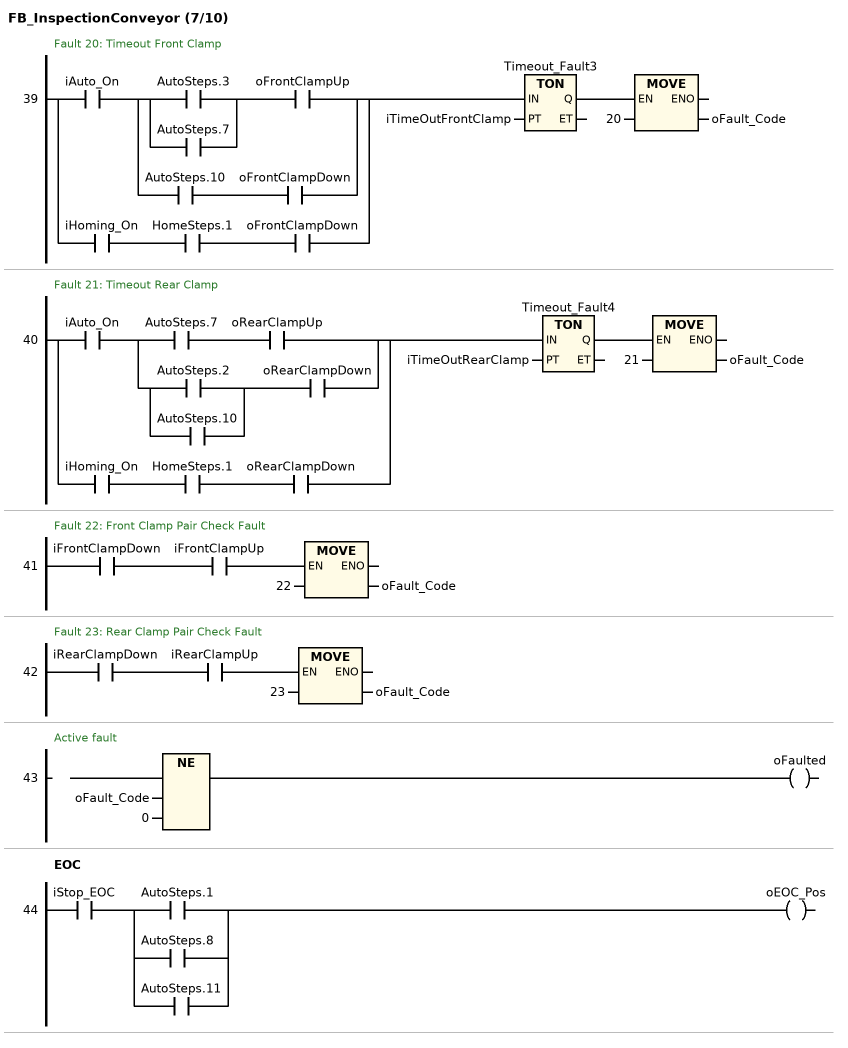
// NETWORK 39
// Fault 20: Timeout Front Clamp
Timeout_Fault3(IN := iAuto_On AND ((AutoSteps.3 OR AutoSteps.7) AND oFrontClampUp OR AutoSteps.10 AND oFrontClampDown) OR iHoming_On AND HomeSteps.1 AND oFrontClampDown, PT := iTimeOutFrontClamp); // TON
IF Timeout_Fault3.Q THEN oFault_Code := 20; END_IF

// NETWORK 40
// Fault 21: Timeout Rear Clamp
Timeout_Fault4(IN := iAuto_On AND (AutoSteps.7 AND oRearClampUp OR (AutoSteps.2 OR AutoSteps.10) AND oRearClampDown) OR iHoming_On AND HomeSteps.1 AND oRearClampDown, PT := iTimeOutRearClamp); // TON
IF Timeout_Fault4.Q THEN oFault_Code := 21; END_IF

// NETWORK 41
// Fault 22: Front Clamp Pair Check Fault
IF iFrontClampDown AND iFrontClampUp THEN oFault_Code := 22; END_IF

// NETWORK 42
// Fault 23: Rear Clamp Pair Check Fault
IF iRearClampDown AND iRearClampUp THEN oFault_Code := 23; END_IF

// NETWORK 43
// Active fault
oFaulted := oFault_Code <> 0;

// NETWORK 44: EOC
oEOC_Pos := iStop_EOC AND (AutoSteps.1 OR AutoSteps.8 OR AutoSteps.11);

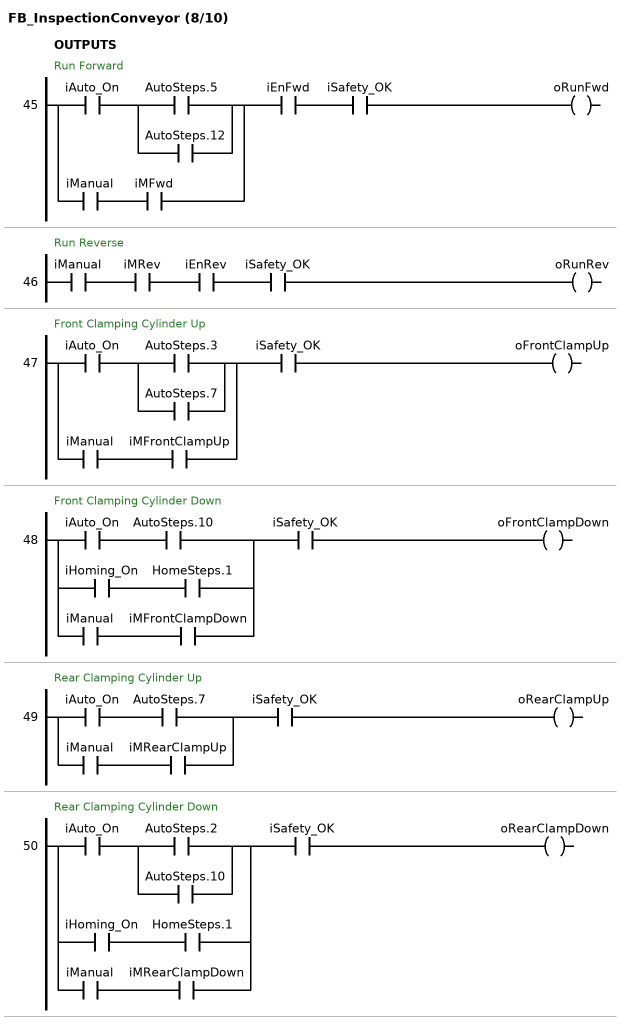
// NETWORK 45: OUTPUTS
// Run Forward
oRunFwd := (iAuto_On AND (AutoSteps.5 OR AutoSteps.12) OR iManual AND iMFwd) AND iEnFwd AND iSafety_OK;

// NETWORK 46
// Run Reverse
oRunRev := iManual AND iMRev AND iEnRev AND iSafety_OK;

// NETWORK 47
// Front Clamping Cylinder Up
oFrontClampUp := (iAuto_On AND (AutoSteps.3 OR AutoSteps.7) OR iManual AND iMFrontClampUp) AND iSafety_OK;

// NETWORK 48
// Front Clamping Cylinder Down
oFrontClampDown := (iAuto_On AND AutoSteps.10 OR iHoming_On AND HomeSteps.1 OR iManual AND iMFrontClampDown) AND iSafety_OK;

// NETWORK 49
// Rear Clamping Cylinder Up
oRearClampUp := (iAuto_On AND AutoSteps.7 OR iManual AND iMRearClampUp) AND iSafety_OK;

// NETWORK 50
// Rear Clamping Cylinder Down
oRearClampDown := (iAuto_On AND (AutoSteps.2 OR AutoSteps.10) OR iHoming_On AND HomeSteps.1 OR iManual AND iMRearClampDown) AND iSafety_OK;

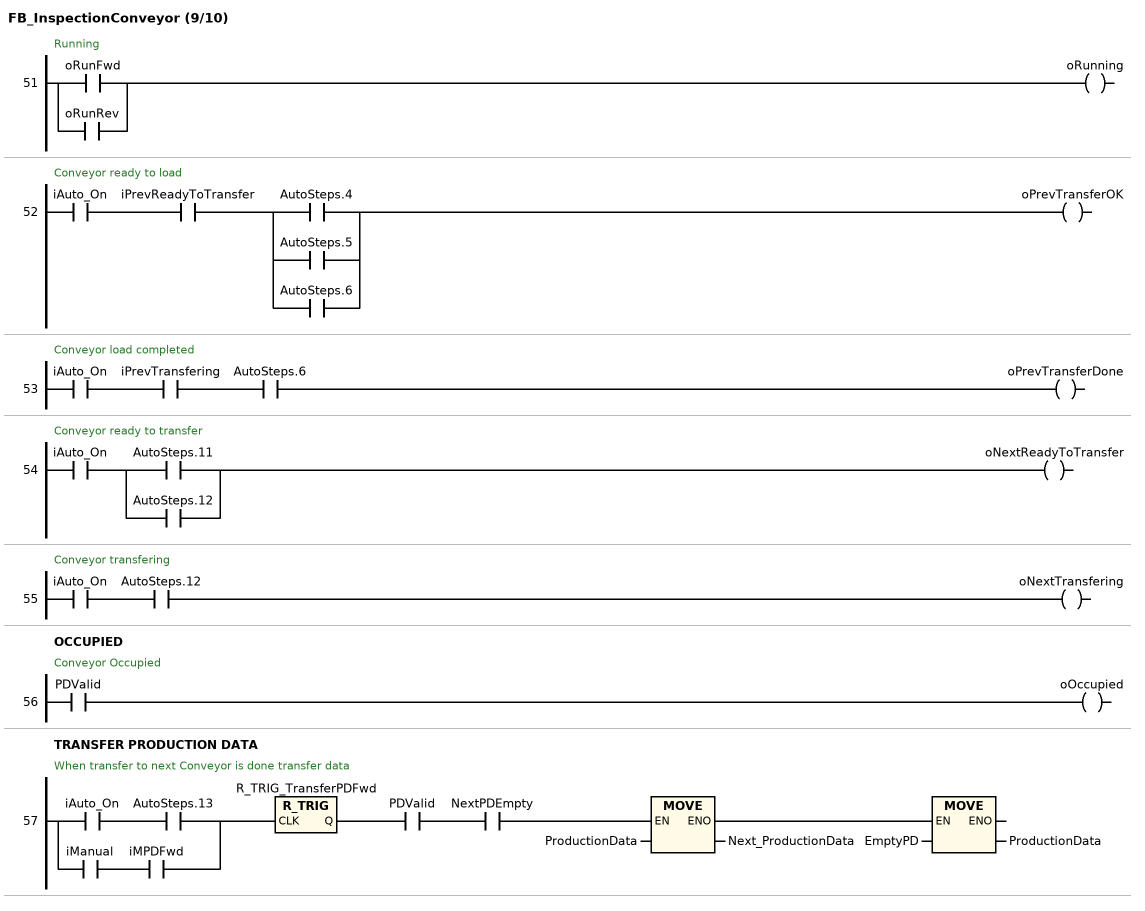
// NETWORK 51
// Running
oRunning := oRunFwd OR oRunRev;

// NETWORK 52
// Conveyor ready to load
oPrevTransferOK := iAuto_On AND iPrevReadyToTransfer AND (AutoSteps.4 OR AutoSteps.5 OR AutoSteps.6);

// NETWORK 53
// Conveyor load completed
oPrevTransferDone := iAuto_On AND iPrevTransfering AND AutoSteps.6;

// NETWORK 54
// Conveyor ready to transfer
oNextReadyToTransfer := iAuto_On AND (AutoSteps.11 OR AutoSteps.12);

// NETWORK 55
// Conveyor transfering
oNextTransfering := iAuto_On AND AutoSteps.12;

// NETWORK 56: OCCUPIED
// Conveyor Occupied
oOccupied := PDValid;

// NETWORK 57: TRANSFER PRODUCTION DATA
// When transfer to next Conveyor is done transfer data
R_TRIG_TransferPDFwd(CLK := iAuto_On AND AutoSteps.13 OR iManual AND iMPDFwd); // R_TRIG
_w20 := R_TRIG_TransferPDFwd.Q AND PDValid AND NextPDEmpty;
IF _w20 THEN Next_ProductionData := ProductionData; END_IF
IF _w20 THEN ProductionData := EmptyPD; END_IF

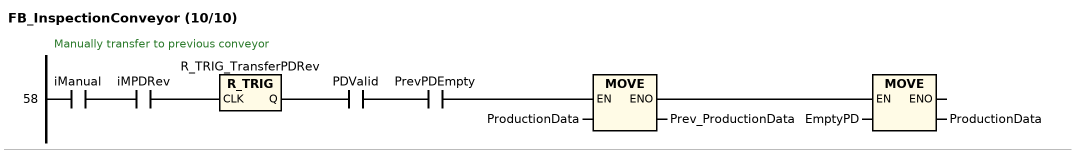
// NETWORK 58
// Manually transfer to previous conveyor
R_TRIG_TransferPDRev(CLK := iManual AND iMPDRev); // R_TRIG
_w21 := R_TRIG_TransferPDRev.Q AND PDValid AND PrevPDEmpty;
IF _w21 THEN Prev_ProductionData := ProductionData; END_IF
IF _w21 THEN ProductionData := EmptyPD; END_IF

END_FUNCTION_BLOCK

// Device/Application/FBs/Convert_RFID
FUNCTION Convert_RFID : STRING
VAR_INPUT
	iLecture: STRING := '';
	iID: UDINT := 0;
	iNumber: UINT := 0;
	iStatus: WORD := 0;
END_VAR
VAR_OUTPUT
	oID: UDINT;
	oNumber: UINT;
	oStatus: WORD;
END_VAR

oID := STRING_TO_UDINT(LEFT(iLecture, 4));
oNumber := STRING_TO_UINT(RIGHT(LEFT(iLecture, 8),4));
oStatus := STRING_TO_WORD(RIGHT(iLecture, 16));


Convert_RFID := CONCAT(UDINT_TO_STRING(iID),CONCAT(UINT_TO_STRING(iNumber),WORD_TO_STRING(iStatus)));

END_FUNCTION

// Device/Application/FBs/CombineData
PROGRAM CombineData
VAR_INPUT
	iCycleTime: STRING(1024);
	iProduct: STRING(1024);
END_VAR
VAR_OUTPUT
	oString: STRING(1024);
END_VAR

oString := CONCAT(iCycleTime,CONCAT('-',iProduct));

END_PROGRAM

// Device/Application/SOP630
PROGRAM SOP630
VAR
END_VAR

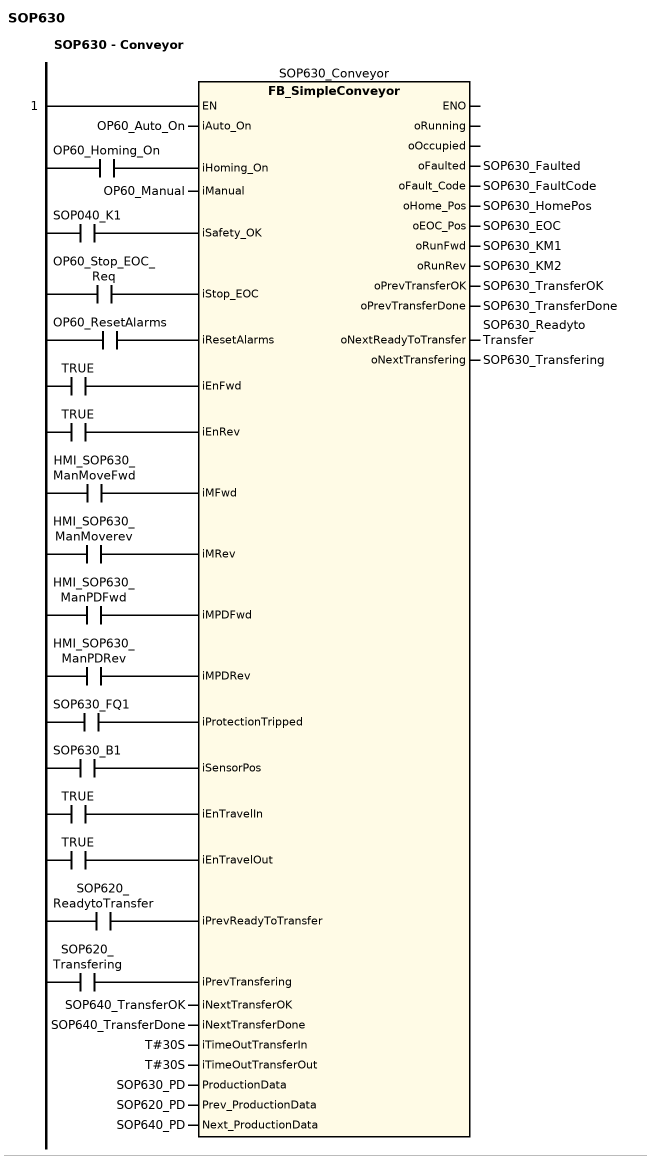
// NETWORK 1: SOP630 - Conveyor
SOP630_Conveyor(
    iAuto_On := OP60_Auto_On,
    iHoming_On := OP60_Homing_On,
    iManual := OP60_Manual,
    iSafety_OK := SOP040_K1,
    iStop_EOC := OP60_Stop_EOC_Req,
    iResetAlarms := OP60_ResetAlarms,
    iEnFwd := TRUE,
    iEnRev := TRUE,
    iMFwd := HMI_SOP630_ManMoveFwd,
    iMRev := HMI_SOP630_ManMoverev,
    iMPDFwd := HMI_SOP630_ManPDFwd,
    iMPDRev := HMI_SOP630_ManPDRev,
    iProtectionTripped := SOP630_FQ1,
    iSensorPos := SOP630_B1,
    iEnTravelIn := TRUE,
    iEnTravelOut := TRUE,
    iPrevReadyToTransfer := SOP620_ReadytoTransfer,
    iPrevTransfering := SOP620_Transfering,
    iNextTransferOK := SOP640_TransferOK,
    iNextTransferDone := SOP640_TransferDone,
    iTimeOutTransferIn := T#30S,
    iTimeOutTransferOut := T#30S,
    ProductionData := SOP630_PD,
    Prev_ProductionData := SOP620_PD,
    Next_ProductionData := SOP640_PD,
    oFaulted => SOP630_Faulted,
    oFault_Code => SOP630_FaultCode,
    oHome_Pos => SOP630_HomePos,
    oEOC_Pos => SOP630_EOC,
    oRunFwd => SOP630_KM1,
    oRunRev => SOP630_KM2,
    oPrevTransferOK => SOP630_TransferOK,
    oPrevTransferDone => SOP630_TransferDone,
    oNextReadyToTransfer => SOP630_ReadytoTransfer,
    oNextTransfering => SOP630_Transfering); // FB_SimpleConveyor

END_PROGRAM

// Device/Application/SOP620
PROGRAM SOP620
VAR
END_VAR

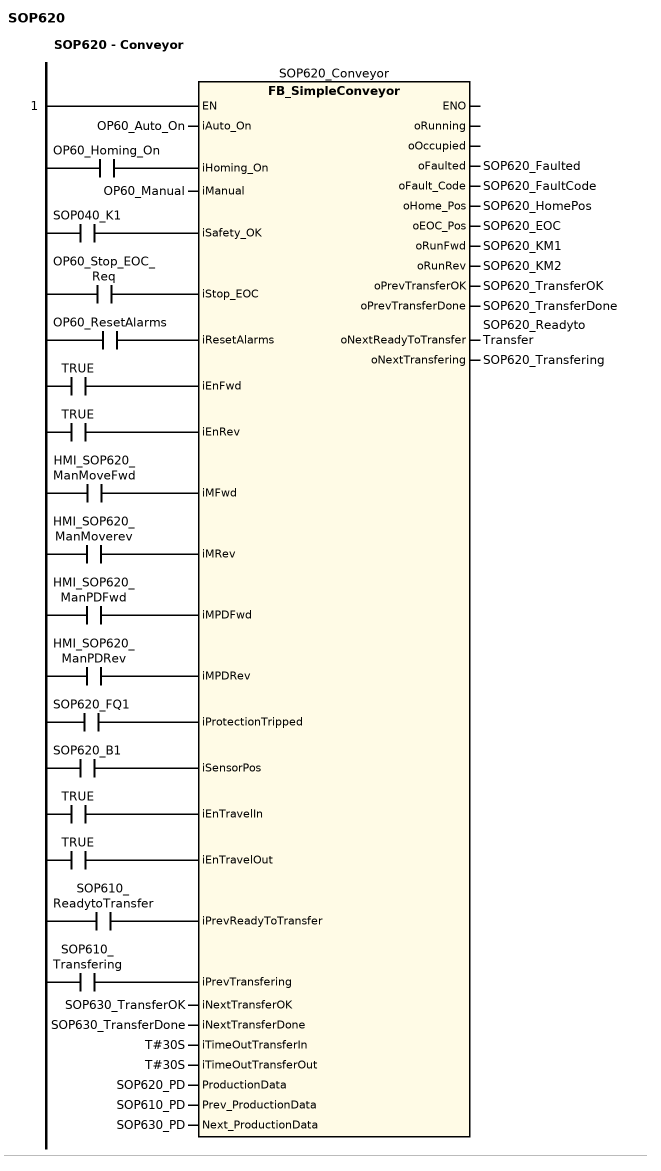
// NETWORK 1: SOP620 - Conveyor
SOP620_Conveyor(
    iAuto_On := OP60_Auto_On,
    iHoming_On := OP60_Homing_On,
    iManual := OP60_Manual,
    iSafety_OK := SOP040_K1,
    iStop_EOC := OP60_Stop_EOC_Req,
    iResetAlarms := OP60_ResetAlarms,
    iEnFwd := TRUE,
    iEnRev := TRUE,
    iMFwd := HMI_SOP620_ManMoveFwd,
    iMRev := HMI_SOP620_ManMoverev,
    iMPDFwd := HMI_SOP620_ManPDFwd,
    iMPDRev := HMI_SOP620_ManPDRev,
    iProtectionTripped := SOP620_FQ1,
    iSensorPos := SOP620_B1,
    iEnTravelIn := TRUE,
    iEnTravelOut := TRUE,
    iPrevReadyToTransfer := SOP610_ReadytoTransfer,
    iPrevTransfering := SOP610_Transfering,
    iNextTransferOK := SOP630_TransferOK,
    iNextTransferDone := SOP630_TransferDone,
    iTimeOutTransferIn := T#30S,
    iTimeOutTransferOut := T#30S,
    ProductionData := SOP620_PD,
    Prev_ProductionData := SOP610_PD,
    Next_ProductionData := SOP630_PD,
    oFaulted => SOP620_Faulted,
    oFault_Code => SOP620_FaultCode,
    oHome_Pos => SOP620_HomePos,
    oEOC_Pos => SOP620_EOC,
    oRunFwd => SOP620_KM1,
    oRunRev => SOP620_KM2,
    oPrevTransferOK => SOP620_TransferOK,
    oPrevTransferDone => SOP620_TransferDone,
    oNextReadyToTransfer => SOP620_ReadytoTransfer,
    oNextTransfering => SOP620_Transfering); // FB_SimpleConveyor

END_PROGRAM

// Device/Application/SOP610
PROGRAM SOP610
VAR
	ID_counter: UDINT := 1000;
	Check_not_empty_msg: BOOL;
END_VAR
VAR // added by the converter: edge detectors and wires of the graphical bodies
    _w1, _w2, _w3, _w4, _w5, _w6, _w7 : BOOL;
    _rt1, _rt2 : R_TRIG;
END_VAR

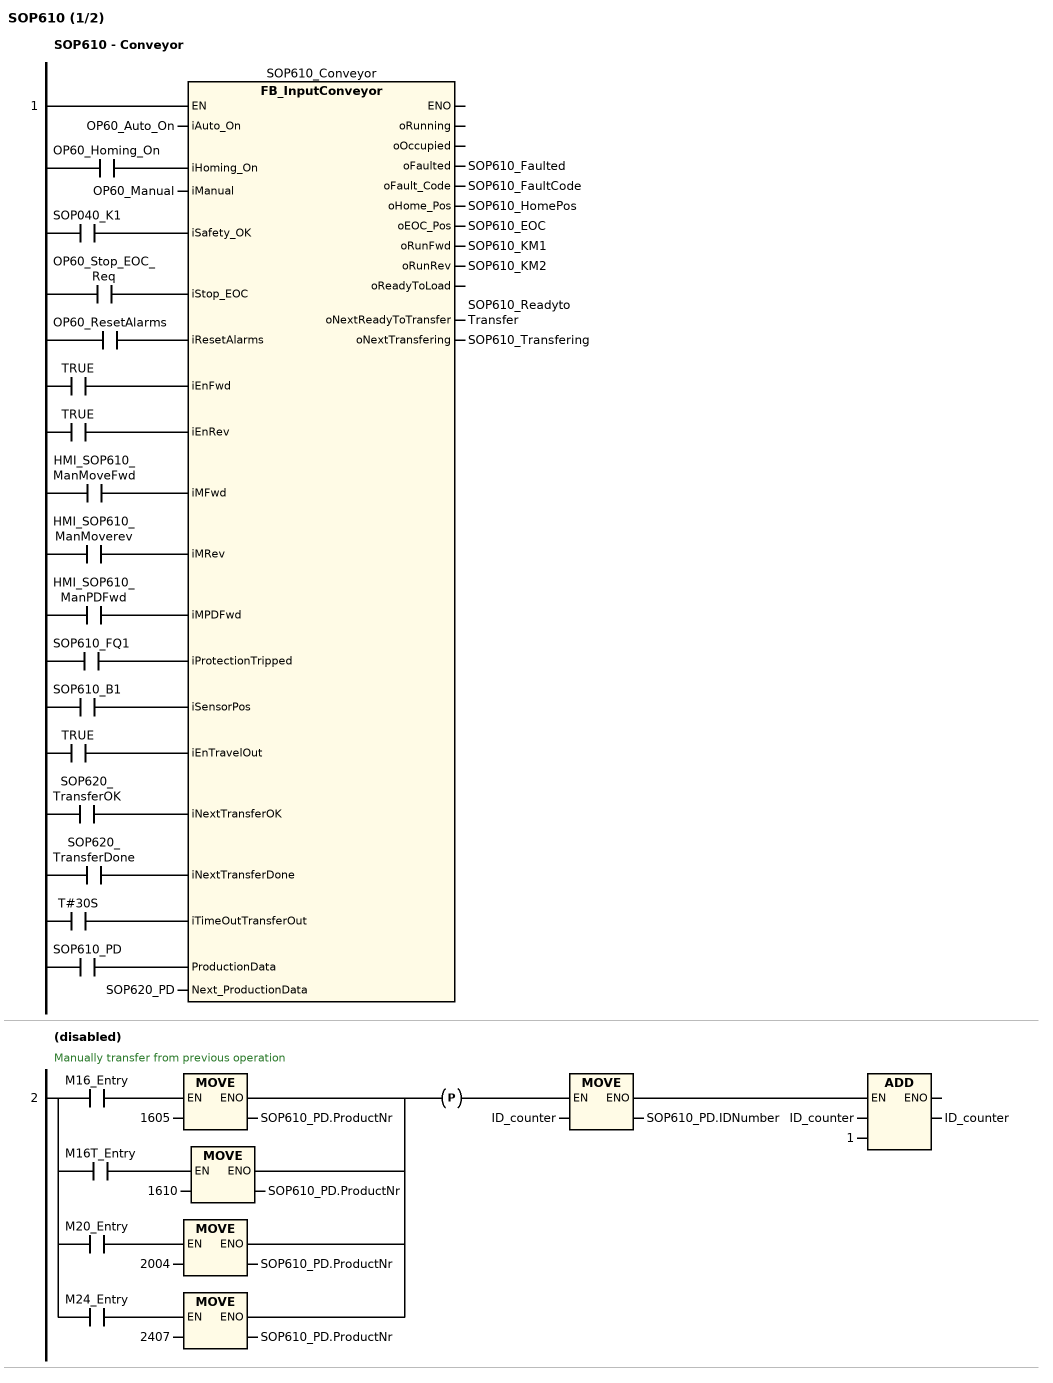
// NETWORK 1: SOP610 - Conveyor
SOP610_Conveyor(
    iAuto_On := OP60_Auto_On,
    iHoming_On := OP60_Homing_On,
    iManual := OP60_Manual,
    iSafety_OK := SOP040_K1,
    iStop_EOC := OP60_Stop_EOC_Req,
    iResetAlarms := OP60_ResetAlarms,
    iEnFwd := TRUE,
    iEnRev := TRUE,
    iMFwd := HMI_SOP610_ManMoveFwd,
    iMRev := HMI_SOP610_ManMoverev,
    iMPDFwd := HMI_SOP610_ManPDFwd,
    iProtectionTripped := SOP610_FQ1,
    iSensorPos := SOP610_B1,
    iEnTravelOut := TRUE,
    iNextTransferOK := SOP620_TransferOK,
    iNextTransferDone := SOP620_TransferDone,
    iTimeOutTransferOut := T#30S,
    ProductionData := SOP610_PD,
    Next_ProductionData := SOP620_PD,
    oFaulted => SOP610_Faulted,
    oFault_Code => SOP610_FaultCode,
    oHome_Pos => SOP610_HomePos,
    oEOC_Pos => SOP610_EOC,
    oRunFwd => SOP610_KM1,
    oRunRev => SOP610_KM2,
    oNextReadyToTransfer => SOP610_ReadytoTransfer,
    oNextTransfering => SOP610_Transfering); // FB_InputConveyor

// NETWORK 2 (disabled)
// Manually transfer from previous operation
// _w1 := M16_Entry;
// IF _w1 THEN SOP610_PD.ProductNr := 1605; END_IF
// _w2 := M16T_Entry;
// IF _w2 THEN SOP610_PD.ProductNr := 1610; END_IF
// _w3 := M20_Entry;
// IF _w3 THEN SOP610_PD.ProductNr := 2004; END_IF
// _w4 := M24_Entry;
// IF _w4 THEN SOP610_PD.ProductNr := 2407; END_IF
// _rt1(CLK := _w1 OR _w2 OR _w3 OR _w4);
// _w5 := _rt1.Q;
// IF _w5 THEN SOP610_PD.IDNumber := ID_counter; END_IF
// IF _w5 THEN ID_counter := ID_counter + 1; END_IF

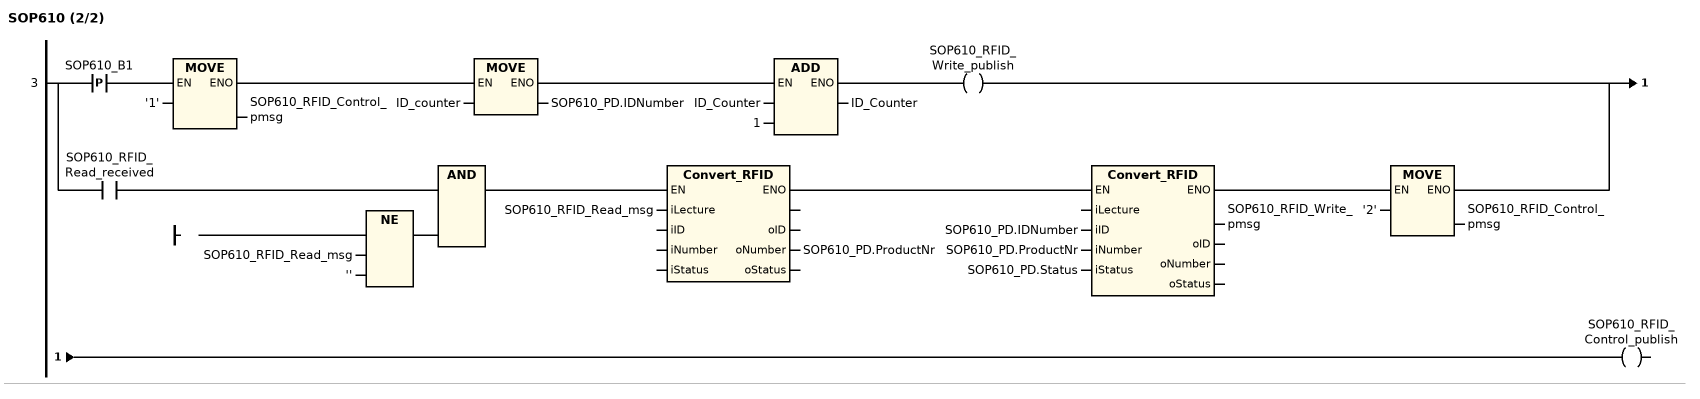
// NETWORK 3
_rt2(CLK := SOP610_B1);
_w6 := _rt2.Q;
IF _w6 THEN SOP610_RFID_Control_pmsg := '1'; END_IF
IF _w6 THEN SOP610_PD.IDNumber := ID_counter; END_IF
IF _w6 THEN ID_Counter := ID_Counter + 1; END_IF
SOP610_RFID_Write_publish := _w6;
_w7 := SOP610_RFID_Read_received AND SOP610_RFID_Read_msg <> '';
IF _w7 THEN Convert_RFID(iLecture := SOP610_RFID_Read_msg, oNumber => SOP610_PD.ProductNr); END_IF
IF _w7 THEN
    SOP610_RFID_Write_pmsg := Convert_RFID(iID := SOP610_PD.IDNumber, iNumber := SOP610_PD.ProductNr, iStatus := SOP610_PD.Status);
END_IF
IF _w7 THEN SOP610_RFID_Control_pmsg := '2'; END_IF
SOP610_RFID_Control_publish := _w6 OR _w7;

END_PROGRAM

// Device/Application/FBs/FB_InputConveyor
FUNCTION_BLOCK FB_InputConveyor
VAR_INPUT
	iAuto_On: BOOL; // Auto-On cycle active
	iHoming_On: BOOL; // Homing-On cycle active
	iManual: BOOL; // Manual mode active
	iSafety_OK: BOOL; // Safety circuit OK
	iStop_EOC: BOOL; // Stop EOC selected
	iResetAlarms: BOOL; // Reset Alarms
	
	iEnFwd: BOOL := TRUE; // Interlock signal movement forward
	iEnRev: BOOL := TRUE; // Interlock signal movement reverse
	
	iMFwd: BOOL; 	// Manual Fwd request
	iMRev: BOOL; 	// Manual Rev request
	iMPDFwd: BOOL; 	// Manual Move PD forward
	
	iProtectionTripped: BOOL := FALSE; // Motor Protection Tripped
	
	iSensorPos: BOOL; // Product in position
	
	iEnTravelOut: BOOL := TRUE; // Enable product transfer to next conveyor.
	
	iNextTransferOK: BOOL; // Next conveyor ready to load
	iNextTransferDone: BOOL;  // Next conveyor transfer done
	
	iTimeOutTransferOut: TIME := T#10S; // Time out time for transfer out
END_VAR
VAR_IN_OUT
	ProductionData: ProductionData; 		// Production Data
	Next_ProductionData: ProductionData;	// Next Production Data
END_VAR
VAR_OUTPUT
	oRunning: BOOL; // Conveyor Running
	oOccupied: BOOL; // Conveyor Occupied
	oFaulted : BOOL; // Conveyor faulted
	oFault_Code: INT; // Conveyor fault code
	oHome_Pos: BOOL; // Conveyor Home Position reached
	oEOC_Pos: BOOL; // Conveyor Stop EOC reached

	oRunFwd: BOOL; // Conveyor running forward
	oRunRev: BOOL; // Conveyor running reverse	

	oReadyToLoad: BOOL; // Conveyor ready to be loaded
	oNextReadyToTransfer: BOOL; // Conveyor ready to transfer
	oNextTransfering: BOOL; // Conveyor transfering
END_VAR
VAR
	AutoSteps: WORD;
	HomeSteps: WORD;
	
	Timeout_Fault2: TON;
	
	EmptyPD: ProductionData;
	PDValid: BOOL;		// PD is Valid
	PDEmpty: BOOL;		// PD is Empty
	NextPDValid: BOOL;	// Next PD is Valid
	NextPDEmpty: BOOL;	// Next PD is Empty
	R_TRIG_TransferPDFwd: R_TRIG;
	R_TRIG_Fault_10: R_TRIG;
	R_TRIG_Fault_12: R_TRIG;
END_VAR
VAR // added by the converter: edge detectors and wires of the graphical bodies
    _w1, _w2, _w3, _w4, _w5, _w6, _w7, _w8, _w9, _w10 : BOOL;
END_VAR

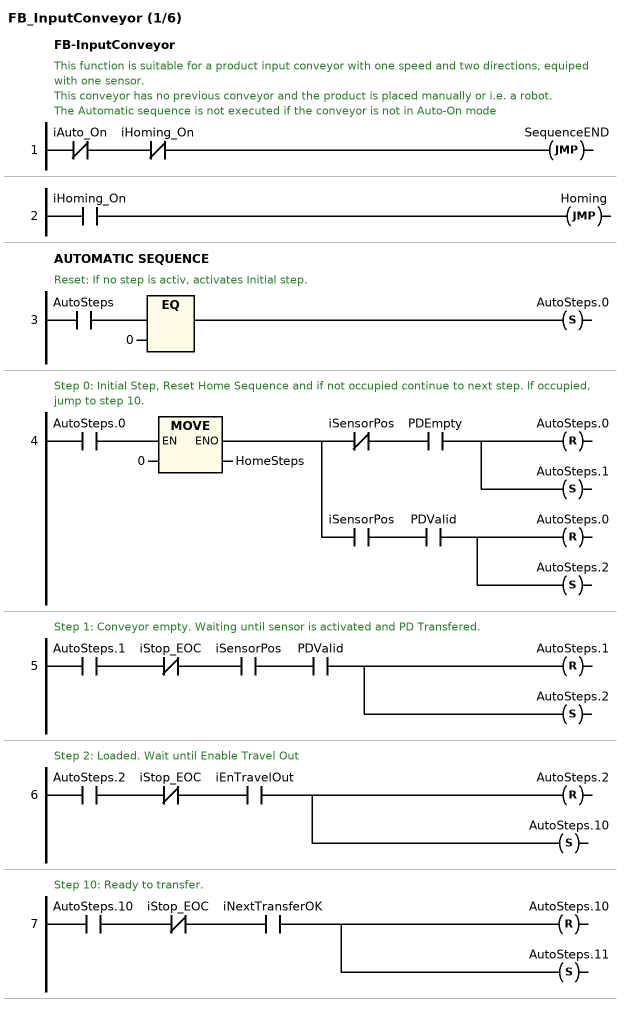
// NETWORK 1: FB-InputConveyor
// This function is suitable for a product input conveyor with one speed and two directions, equiped with one sensor.
// This conveyor has no previous conveyor and the product is placed manually or i.e. a robot.
// The Automatic sequence is not executed if the conveyor is not in Auto-On mode
IF NOT iAuto_On AND NOT iHoming_On THEN JMP SequenceEND; END_IF

// NETWORK 2
IF iHoming_On THEN JMP Homing; END_IF

// NETWORK 3: AUTOMATIC SEQUENCE
// Reset: If no step is activ, activates Initial step.
AutoSteps.0 S= AutoSteps = 0;

// NETWORK 4
// Step 0: Initial Step, Reset Home Sequence and if not occupied continue to next step. If occupied, jump to step 10.
_w1 := AutoSteps.0;
IF _w1 THEN HomeSteps := 0; END_IF
_w2 := _w1 AND NOT iSensorPos AND PDEmpty;
AutoSteps.0 R= _w2;
AutoSteps.1 S= _w2;
_w3 := _w1 AND iSensorPos AND PDValid;
AutoSteps.0 R= _w3;
AutoSteps.2 S= _w3;

// NETWORK 5
// Step 1: Conveyor empty. Waiting until sensor is activated and PD Transfered.
_w4 := AutoSteps.1 AND NOT iStop_EOC AND iSensorPos AND PDValid;
AutoSteps.1 R= _w4;
AutoSteps.2 S= _w4;

// NETWORK 6
// Step 2: Loaded. Wait until Enable Travel Out
_w5 := AutoSteps.2 AND NOT iStop_EOC AND iEnTravelOut;
AutoSteps.2 R= _w5;
AutoSteps.10 S= _w5;

// NETWORK 7
// Step 10: Ready to transfer.
_w6 := AutoSteps.10 AND NOT iStop_EOC AND iNextTransferOK;
AutoSteps.10 R= _w6;
AutoSteps.11 S= _w6;

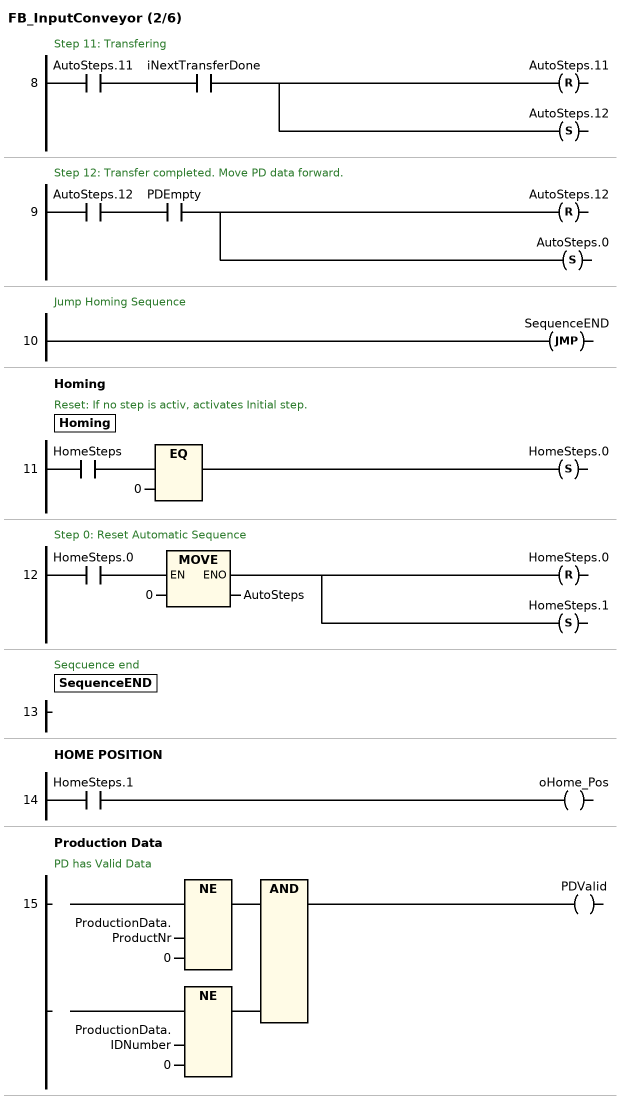
// NETWORK 8
// Step 11: Transfering
_w7 := AutoSteps.11 AND iNextTransferDone;
AutoSteps.11 R= _w7;
AutoSteps.12 S= _w7;

// NETWORK 9
// Step 12: Transfer completed. Move PD data forward.
_w8 := AutoSteps.12 AND PDEmpty;
AutoSteps.12 R= _w8;
AutoSteps.0 S= _w8;

// NETWORK 10
// Jump Homing Sequence
JMP SequenceEND;

// NETWORK 11: Homing
// Reset: If no step is activ, activates Initial step.
Homing:
HomeSteps.0 S= HomeSteps = 0;

// NETWORK 12
// Step 0: Reset Automatic Sequence
_w9 := HomeSteps.0;
IF _w9 THEN AutoSteps := 0; END_IF
HomeSteps.0 R= _w9;
HomeSteps.1 S= _w9;

// NETWORK 13
// Seqcuence end
SequenceEND: ;

// NETWORK 14: HOME POSITION
oHome_Pos := HomeSteps.1;

// NETWORK 15: Production Data
// PD has Valid Data
PDValid := ProductionData.ProductNr <> 0 AND ProductionData.IDNumber <> 0;

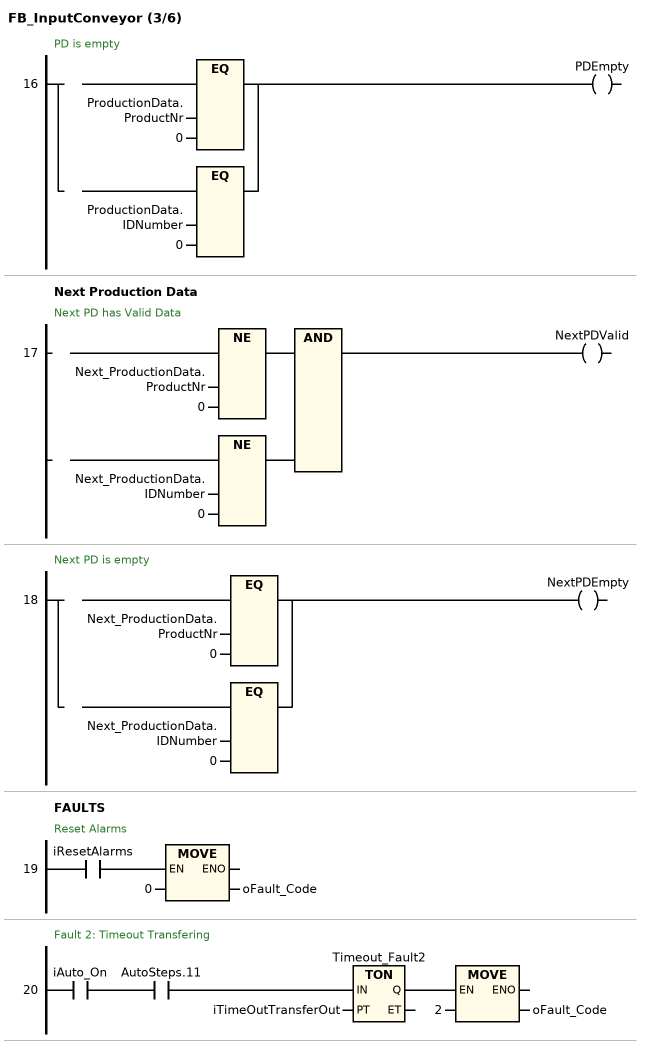
// NETWORK 16
// PD is empty
PDEmpty := ProductionData.ProductNr = 0 OR ProductionData.IDNumber = 0;

// NETWORK 17: Next Production Data
// Next PD has Valid Data
NextPDValid := Next_ProductionData.ProductNr <> 0 AND Next_ProductionData.IDNumber <> 0;

// NETWORK 18
// Next PD is empty
NextPDEmpty := Next_ProductionData.ProductNr = 0 OR Next_ProductionData.IDNumber = 0;

// NETWORK 19: FAULTS
// Reset Alarms
IF iResetAlarms THEN oFault_Code := 0; END_IF

// NETWORK 20
// Fault 2: Timeout Transfering
Timeout_Fault2(IN := iAuto_On AND AutoSteps.11, PT := iTimeOutTransferOut); // TON
IF Timeout_Fault2.Q THEN oFault_Code := 2; END_IF

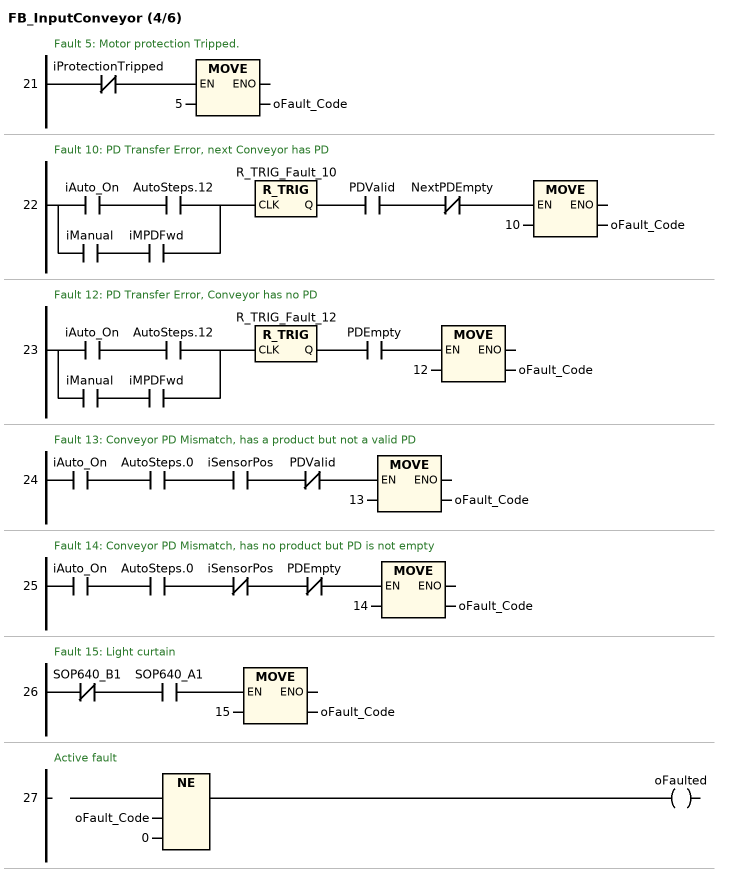
// NETWORK 21
// Fault 5: Motor protection Tripped.
IF NOT iProtectionTripped THEN oFault_Code := 5; END_IF

// NETWORK 22
// Fault 10: PD Transfer Error, next Conveyor has PD
R_TRIG_Fault_10(CLK := iAuto_On AND AutoSteps.12 OR iManual AND iMPDFwd); // R_TRIG
IF R_TRIG_Fault_10.Q AND PDValid AND NOT NextPDEmpty THEN oFault_Code := 10; END_IF

// NETWORK 23
// Fault 12: PD Transfer Error, Conveyor has no PD
R_TRIG_Fault_12(CLK := iAuto_On AND AutoSteps.12 OR iManual AND iMPDFwd); // R_TRIG
IF R_TRIG_Fault_12.Q AND PDEmpty THEN oFault_Code := 12; END_IF

// NETWORK 24
// Fault 13: Conveyor PD Mismatch, has a product but not a valid PD
IF iAuto_On AND AutoSteps.0 AND iSensorPos AND NOT PDValid THEN oFault_Code := 13; END_IF

// NETWORK 25
// Fault 14: Conveyor PD Mismatch, has no product but PD is not empty
IF iAuto_On AND AutoSteps.0 AND NOT iSensorPos AND NOT PDEmpty THEN oFault_Code := 14; END_IF

// NETWORK 26
// Fault 15: Light curtain
IF NOT SOP640_B1 AND SOP640_A1 THEN oFault_Code := 15; END_IF

// NETWORK 27
// Active fault
oFaulted := oFault_Code <> 0;

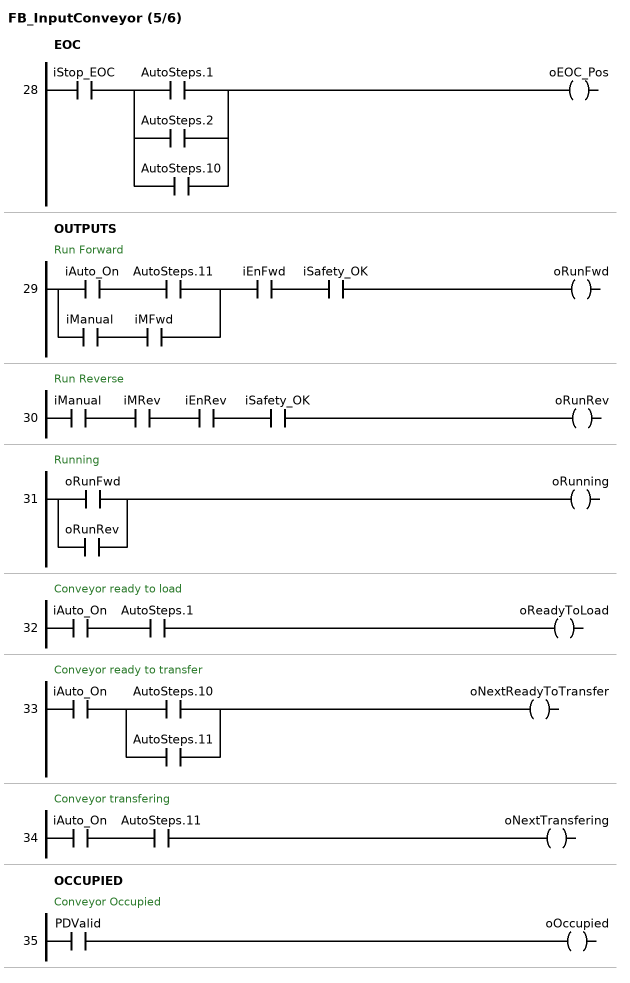
// NETWORK 28: EOC
oEOC_Pos := iStop_EOC AND (AutoSteps.1 OR AutoSteps.2 OR AutoSteps.10);

// NETWORK 29: OUTPUTS
// Run Forward
oRunFwd := (iAuto_On AND AutoSteps.11 OR iManual AND iMFwd) AND iEnFwd AND iSafety_OK;

// NETWORK 30
// Run Reverse
oRunRev := iManual AND iMRev AND iEnRev AND iSafety_OK;

// NETWORK 31
// Running
oRunning := oRunFwd OR oRunRev;

// NETWORK 32
// Conveyor ready to load
oReadyToLoad := iAuto_On AND AutoSteps.1;

// NETWORK 33
// Conveyor ready to transfer
oNextReadyToTransfer := iAuto_On AND (AutoSteps.10 OR AutoSteps.11);

// NETWORK 34
// Conveyor transfering
oNextTransfering := iAuto_On AND AutoSteps.11;

// NETWORK 35: OCCUPIED
// Conveyor Occupied
oOccupied := PDValid;

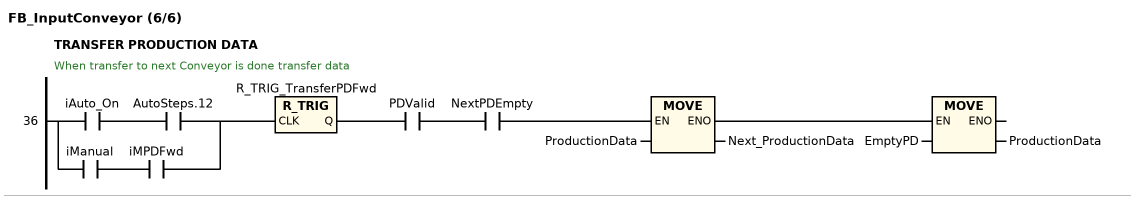
// NETWORK 36: TRANSFER PRODUCTION DATA
// When transfer to next Conveyor is done transfer data
R_TRIG_TransferPDFwd(CLK := iAuto_On AND AutoSteps.12 OR iManual AND iMPDFwd); // R_TRIG
_w10 := R_TRIG_TransferPDFwd.Q AND PDValid AND NextPDEmpty;
IF _w10 THEN Next_ProductionData := ProductionData; END_IF
IF _w10 THEN ProductionData := EmptyPD; END_IF

END_FUNCTION_BLOCK

// Device/Application/SOP600
PROGRAM SOP600
VAR
END_VAR

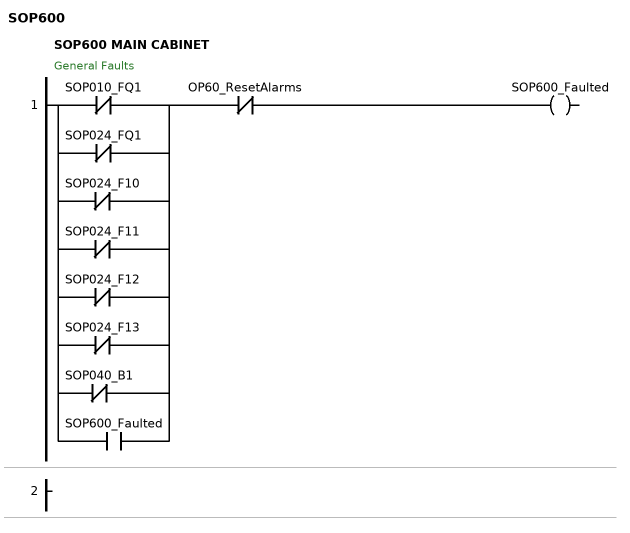
// NETWORK 1: SOP600 MAIN CABINET
// General Faults
SOP600_Faulted := (NOT SOP010_FQ1 OR NOT SOP024_FQ1 OR NOT SOP024_F10 OR NOT SOP024_F11 OR NOT SOP024_F12 OR NOT SOP024_F13 OR NOT SOP040_B1 OR SOP600_Faulted) AND NOT OP60_ResetAlarms;

// NETWORK 2

END_PROGRAM

// Device/Application/MQTT_Sensors_Actuators
PROGRAM MQTT_Sensors_Actuators
VAR
	// MQTT BROKER INFORMATION
		MQTTClient: MQTT.MQTTClient; 										// MQTTClient FB
		MQTTClient1: MQTT.MQTTClient;										// MQTTClient FB
		MQTTClient2: MQTT.MQTTClient;										// MQTTClient FB
		MQTTClient3: MQTT.MQTTClient;										// MQTTClient FB
		MQTTClient4: MQTT.MQTTClient;										// MQTTClient FB
		
		Port: UINT := 1883; 												// Port
		Will_msg: STRING(1024) := ''; 										// Message if there is disconnection
		Host: STRING(255) := '192.168.1.123'; 								// Broker IP 192.168.1.123 Simumatik
		Codesys: WSTRING(1024) := "codesys";								// Username and password "Codesys"
		
		Enable_Client: BOOL := TRUE; 										// Establishes connecting with the MQTT broker
	
	// SOP640 INSPECTION SUBSCRIPTION
		MQTTSubscribe_SOP640: MQTT.MQTTSubscribe;						 		// MQTTSubscribe FB
		SOP640_Topic: WSTRING(1024) := "OP60/SOP640/Inspection"; 					// Topic SOP640
		
	// SOP640 PRESSENCE PUBLISH
		MQTTPublish_SOP640: MQTT.MQTTPublish;									// MQTTPublish FB
		SOP640_pTopic: WSTRING(1024) := "OP60/Alarms";							// Topic pALARMS
	
	// Schedule SUBSCRIPTION
		MQTTSubscribe_Schedule_Start: MQTT.MQTTSubscribe;					// MQTTSubscribe FB
		Schedule_Start_Topic: WSTRING(1024) := "OP60/Schedule/Start";				// Topic Schedule
		
	// Schedule PUBLISH
		MQTTSubscribe_Schedule_End: MQTT.MQTTSubscribe;						// MQTTPublish FB
		Schedule_End_Topic: WSTRING(1024) := "OP60/Schedule/End";				// Topic pSchedule
	
	// Lights SUBSCRIPTION/PUBLISH
		MQTTSubscribe_Illumination: MQTT.MQTTSubscribe;								// MQTT Subscribe FB
		Illumination_Topic: WSTRING(1024) := "OP60/Illumination";					// Topic Illumination
		MQTTPublish_Illumination: MQTT.MQTTPublish;									// MQTT Publish FB
		
	// Cycle Data PUBLISH
		MQTTPublish_CycleData: MQTT.MQTTPublish;								// MQTTPublish FB
		CycleData_pTopic: WSTRING(1024):= "OP60/CycleData";						// Topic pCycleData
		
	// Products PUBLISH
		MQTTPublish_Products: MQTT.MQTTPublish;									// MQTTPublish FB
		Products_pTopic: WSTRING(1024):= "OP60/Products";						// Topic pProducts
		
	// Sensors SUBSCRIBE
		MQTTSubscribe_Operator_fault: MQTT.MQTTSubscribe;							// MQTTSubscribe FB
		MQTTSubscribe_SOP010_FQ1: MQTT.MQTTSubscribe;								// MQTTSubscribe FB
		MQTTSubscribe_SOP040_K1: MQTT.MQTTSubscribe;								// MQTTSubscribe FB
		MQTTSubscribe_SOP024_FQ1: MQTT.MQTTSubscribe;								// MQTTSubscribe FB
		MQTTSubscribe_SOP024_F10: MQTT.MQTTSubscribe;								// MQTTSubscribe FB
		MQTTSubscribe_SOP024_F11: MQTT.MQTTSubscribe;								// MQTTSubscribe FB
		MQTTSubscribe_SOP024_F12: MQTT.MQTTSubscribe;								// MQTTSubscribe FB
		MQTTSubscribe_SOP024_F13: MQTT.MQTTSubscribe;								// MQTTSubscribe FB
		MQTTSubscribe_SOP040_B1: MQTT.MQTTSubscribe;								// MQTTSubscribe FB
		MQTTSubscribe_SOP600_S1: MQTT.MQTTSubscribe;								// MQTTSubscribe FB
		MQTTSubscribe_SOP600_S2: MQTT.MQTTSubscribe;								// MQTTSubscribe FB
		MQTTSubscribe_SOP600_S3_4: MQTT.MQTTSubscribe;								// MQTTSubscribe FB
		MQTTSubscribe_SOP600_S5: MQTT.MQTTSubscribe;								// MQTTSubscribe FB
		MQTTSubscribe_SOP600_S6: MQTT.MQTTSubscribe;								// MQTTSubscribe FB
		MQTTSubscribe_SOP600_S7: MQTT.MQTTSubscribe;								// MQTTSubscribe FB
		MQTTSubscribe_SOP600_S8: MQTT.MQTTSubscribe;								// MQTTSubscribe FB
		MQTTSubscribe_SOP600_S9: MQTT.MQTTSubscribe;								// MQTTSubscribe FB
		MQTTSubscribe_SOP600_S10: MQTT.MQTTSubscribe;								// MQTTSubscribe FB
		MQTTSubscribe_SOP600_S11: MQTT.MQTTSubscribe;								// MQTTSubscribe FB
		MQTTSubscribe_SOP610_RFID_Read_Topic: MQTT.MQTTSubscribe;					// MQTTSubscribe FB
		MQTTSubscribe_SOP610_RFID_Status_Topic: MQTT.MQTTSubscribe;					// MQTTSubscribe FB
		MQTTSubscribe_SOP610_B1: MQTT.MQTTSubscribe;								// MQTTSubscribe FB
		MQTTSubscribe_SOP610_FQ1: MQTT.MQTTSubscribe;								// MQTTSubscribe FB
		MQTTSubscribe_SOP620_B1: MQTT.MQTTSubscribe;								// MQTTSubscribe FB
		MQTTSubscribe_SOP620_FQ1: MQTT.MQTTSubscribe;								// MQTTSubscribe FB
		MQTTSubscribe_SOP630_B1: MQTT.MQTTSubscribe;								// MQTTSubscribe FB
		MQTTSubscribe_SOP630_FQ1: MQTT.MQTTSubscribe;								// MQTTSubscribe FB
		MQTTSubscribe_SOP690_RFID_Read_Topic: MQTT.MQTTSubscribe;					// MQTTSubscribe FB
		MQTTSubscribe_SOP690_RFID_Status_Topic: MQTT.MQTTSubscribe;					// MQTTSubscribe FB
		MQTTSubscribe_SOP640_A1: MQTT.MQTTSubscribe;								// MQTTSubscribe FB
		MQTTSubscribe_SOP640_B1: MQTT.MQTTSubscribe;								// MQTTSubscribe FB
		MQTTSubscribe_SOP640_B2: MQTT.MQTTSubscribe;								// MQTTSubscribe FB
		MQTTSubscribe_SOP640_B3: MQTT.MQTTSubscribe;								// MQTTSubscribe FB
		MQTTSubscribe_SOP640_B4: MQTT.MQTTSubscribe;								// MQTTSubscribe FB
		MQTTSubscribe_SOP640_B5: MQTT.MQTTSubscribe;								// MQTTSubscribe FB
		MQTTSubscribe_SOP640_B6: MQTT.MQTTSubscribe;								// MQTTSubscribe FB
		MQTTSubscribe_SOP640_FQ1: MQTT.MQTTSubscribe;								// MQTTSubscribe FB
		MQTTSubscribe_SOP650_B1: MQTT.MQTTSubscribe;								// MQTTSubscribe FB
		MQTTSubscribe_SOP650_FQ1: MQTT.MQTTSubscribe;								// MQTTSubscribe FB
		MQTTSubscribe_SOP660_B1: MQTT.MQTTSubscribe;								// MQTTSubscribe FB
		MQTTSubscribe_SOP660_FQ1: MQTT.MQTTSubscribe;								// MQTTSubscribe FB
		MQTTSubscribe_SOP670_B1: MQTT.MQTTSubscribe;								// MQTTSubscribe FB
		MQTTSubscribe_SOP670_FQ1: MQTT.MQTTSubscribe;								// MQTTSubscribe FB
		MQTTSubscribe_SOP680_B1: MQTT.MQTTSubscribe;								// MQTTSubscribe FB
		MQTTSubscribe_SOP680_FQ1: MQTT.MQTTSubscribe;								// MQTTSubscribe FB
		MQTTSubscribe_SOP690_S1: MQTT.MQTTSubscribe;								// MQTTSubscribe FB
		MQTTSubscribe_SOP690_S2: MQTT.MQTTSubscribe;								// MQTTSubscribe FB
		MQTTSubscribe_SOP690_S3: MQTT.MQTTSubscribe;								// MQTTSubscribe FB
		MQTTSubscribe_SOP690_S4: MQTT.MQTTSubscribe;								// MQTTSubscribe FB
		
		SOP010_FQ1_Topic: WSTRING(1024):= "OP60/Sensor/SOP010_FQ1";						// Topic Sensor SOP010_FQ1
		SOP040_K1_Topic: WSTRING(1024):= "OP60/Sensor/SOP040_K1";						// Topic Sensor SOP040_K1
		SOP024_FQ1_Topic: WSTRING(1024):= "OP60/Sensor/SOP024_FQ1";						// Topic Sensor SOP024_FQ1
		SOP024_F10_Topic: WSTRING(1024):= "OP60/Sensor/SOP024_F10";						// Topic Sensor SOP024_F10
		SOP024_F11_Topic: WSTRING(1024):= "OP60/Sensor/SOP024_F11";						// Topic Sensor SOP024_F11
		SOP024_F12_Topic: WSTRING(1024):= "OP60/Sensor/SOP024_F12";						// Topic Sensor SOP024_F12
		SOP024_F13_Topic: WSTRING(1024):= "OP60/Sensor/SOP024_F13";						// Topic Sensor SOP024_F13
		SOP040_B1_Topic: WSTRING(1024):= "OP60/Sensor/SOP040_B1";						// Topic Sensor SOP040_B1
		SOP600_S1_Topic: WSTRING(1024):= "OP60/Sensor/SOP600_S1";						// Topic Sensor SOP600_S1
		SOP600_S2_Topic: WSTRING(1024):= "OP60/Sensor/SOP600_S2";						// Topic Sensor SOP600_S2
		SOP600_S3_4_Topic: WSTRING(1024):= "OP60/Sensor/SOP600_S3_4";					// Topic Sensor SOP600_S3_4
		SOP600_S5_Topic: WSTRING(1024):= "OP60/Sensor/SOP600_S5";						// Topic Sensor SOP600_S5
		SOP600_S6_Topic: WSTRING(1024):= "OP60/Sensor/SOP600_S6";						// Topic Sensor SOP600_S6
		SOP600_S7_Topic: WSTRING(1024):= "OP60/Sensor/SOP600_S7";						// Topic Sensor SOP600_S7
		SOP600_S8_Topic: WSTRING(1024):= "OP60/Sensor/SOP600_S8";						// Topic Sensor SOP600_S8
		SOP600_S9_Topic: WSTRING(1024):= "OP60/Sensor/SOP600_S9";						// Topic Sensor SOP600_S9
		SOP600_S10_Topic: WSTRING(1024):= "OP60/Sensor/SOP600_S10";						// Topic Sensor SOP600_S10
		SOP600_S11_Topic: WSTRING(1024):= "OP60/Sensor/SOP600_S11";						// Topic Sensor SOP600_S11
		SOP610_RFID_Read_Topic: WSTRING(1024):= "OP60/SOP610/RFID_Read";				// Topic RFID Read
		SOP610_RFID_Status_Topic: WSTRING(1024):= "OP60/SOP610/RFID_Status";			// Topic RFID Status
		SOP610_B1_Topic: WSTRING(1024):= "OP60/Sensor/SOP610_B1";						// Topic Sensor SOP610_B1
		SOP610_FQ1_Topic: WSTRING(1024):= "OP60/Sensor/SOP610_FQ1";						// Topic Sensor SOP610_FQ1
		SOP620_B1_Topic: WSTRING(1024):= "OP60/Sensor/SOP620_B1";						// Topic Sensor SOP620_B1
		SOP620_FQ1_Topic: WSTRING(1024):= "OP60/Sensor/SOP620_FQ1";						// Topic Sensor SOP620_FQ1
		SOP630_B1_Topic: WSTRING(1024):= "OP60/Sensor/SOP630_B1";						// Topic Sensor SOP630_B1
		SOP630_FQ1_Topic: WSTRING(1024):= "OP60/Sensor/SOP630_FQ1";						// Topic Sensor SOP630_FQ1
		SOP690_RFID_Read_Topic: WSTRING(1024):= "OP60/SOP690/RFID_Read";				// Topic RFID Read
		SOP690_RFID_Status_Topic: WSTRING(1024):= "OP60/SOP690/RFID_Status";			// Topic RFID Status
		SOP640_A1_Topic: WSTRING(1024):= "OP60/Sensor/SOP640_A1";						// Topic Sensor SOP640_A1
		SOP640_B1_Topic: WSTRING(1024):= "OP60/Sensor/SOP640_B1";						// Topic Sensor SOP640_B1
		SOP640_B2_Topic: WSTRING(1024):= "OP60/Sensor/SOP640_B2";						// Topic Sensor SOP640_B2
		SOP640_B3_Topic: WSTRING(1024):= "OP60/Sensor/SOP640_B3";						// Topic Sensor SOP640_B3
		SOP640_B4_Topic: WSTRING(1024):= "OP60/Sensor/SOP640_B4";						// Topic Sensor SOP640_B4
		SOP640_B5_Topic: WSTRING(1024):= "OP60/Sensor/SOP640_B5";						// Topic Sensor SOP640_B5
		SOP640_B6_Topic: WSTRING(1024):= "OP60/Sensor/SOP640_B6";						// Topic Sensor SOP640_B6
		SOP640_FQ1_Topic: WSTRING(1024):= "OP60/Sensor/SOP640_FQ1";						// Topic Sensor SOP640_FQ1
		SOP650_B1_Topic: WSTRING(1024):= "OP60/Sensor/SOP650_B1";						// Topic Sensor SOP650_B1
		SOP650_FQ1_Topic: WSTRING(1024):= "OP60/Sensor/SOP650_FQ1";						// Topic Sensor SOP650_FQ1
		SOP660_B1_Topic: WSTRING(1024):= "OP60/Sensor/SOP660_B1";						// Topic Sensor SOP660_B1
		SOP660_FQ1_Topic: WSTRING(1024):= "OP60/Sensor/SOP660_FQ1";						// Topic Sensor SOP660_FQ1
		SOP670_B1_Topic: WSTRING(1024):= "OP60/Sensor/SOP670_B1";						// Topic Sensor SOP670_B1
		SOP670_FQ1_Topic: WSTRING(1024):= "OP60/Sensor/SOP670_FQ1";						// Topic Sensor SOP670_FQ1
		SOP680_B1_Topic: WSTRING(1024):= "OP60/Sensor/SOP680_B1";						// Topic Sensor SOP680_B1
		SOP680_FQ1_Topic: WSTRING(1024):= "OP60/Sensor/SOP680_FQ1";						// Topic Sensor SOP680_FQ1
		SOP690_S1_Topic: WSTRING(1024):= "OP60/Sensor/SOP690_S1";						// Topic Sensor SOP690_S1
		SOP690_S2_Topic: WSTRING(1024):= "OP60/Sensor/SOP690_S2";						// Topic Sensor SOP690_S2
		SOP690_S3_Topic: WSTRING(1024):= "OP60/Sensor/SOP690_S3";						// Topic Sensor SOP690_S3
		SOP690_S4_Topic: WSTRING(1024):= "OP60/Sensor/SOP690_S4";						// Topic Sensor SOP690_S4
		Operator_Fault_Topic: WSTRING(1024) := "OP60/Operator/Fault";					// Topic operator Fault
		
	Enable_Subscribe: BOOL;														// Establishes subscription to topic if TRUE
	Enable_Subscribe1: BOOL;													// Establishes subscription to topic if TRUE
	Enable_Subscribe2: BOOL;													// Establishes subscription to topic if TRUE
	Enable_Subscribe3: BOOL;													// Establishes subscription to topic if TRUE
	Enable_Subscribe4: BOOL;													// Establishes subscription to topic if TRUE
		
	// ACTUATORS PUBLISH
		MQTTPublish_SOP040_K3: MQTT.MQTTPublish;									// MQTTPublish FB
		MQTTPublish_SOP600_H6: MQTT.MQTTPublish;									// MQTTPublish FB
		MQTTPublish_SOP600_H7: MQTT.MQTTPublish;									// MQTTPublish FB
		MQTTPublish_SOP600_H8: MQTT.MQTTPublish;									// MQTTPublish FB
		MQTTPublish_SOP600_H9: MQTT.MQTTPublish;									// MQTTPublish FB
		MQTTPublish_SOP600_S1: MQTT.MQTTPublish;									// MQTTPublish FB
		MQTTPublish_SOP600_S2: MQTT.MQTTPublish;									// MQTTPublish FB
		MQTTPublish_SOP600_S5: MQTT.MQTTPublish;									// MQTTPublish FB
		MQTTPublish_SOP600_S6: MQTT.MQTTPublish;									// MQTTPublish FB
		MQTTPublish_SOP600_S7: MQTT.MQTTPublish;									// MQTTPublish FB
		MQTTPublish_SOP600_S8: MQTT.MQTTPublish;									// MQTTPublish FB
		MQTTPublish_SOP600_S9: MQTT.MQTTPublish;									// MQTTPublish FB
		MQTTPublish_SOP600_S10: MQTT.MQTTPublish;									// MQTTPublish FB
		MQTTPublish_SOP600_S11: MQTT.MQTTPublish;									// MQTTPublish FB
		MQTTPublish_SOP610_RFID_Control: MQTT.MQTTPublish;							// MQTTPublish FB
		MQTTPublish_SOP610_RFID_Write: MQTT.MQTTPublish;							// MQTTPublish FB
		MQTTPublish_SOP610_KM1_2: MQTT.MQTTPublish;									// MQTTPublish FB
		MQTTPublish_SOP620_KM1_2: MQTT.MQTTPublish;									// MQTTPublish FB
		MQTTPublish_SOP630_KM1_2: MQTT.MQTTPublish;									// MQTTPublish FB
		MQTTPublish_SOP640_KM1_2: MQTT.MQTTPublish;									// MQTTPublish FB
		MQTTPublish_SOP640_K2: MQTT.MQTTPublish;									// MQTTPublish FB
		MQTTPublish_SOP640_Y1: MQTT.MQTTPublish;									// MQTTPublish FB
		MQTTPublish_SOP640_Y2: MQTT.MQTTPublish;									// MQTTPublish FB
		MQTTPublish_SOP640_Y3: MQTT.MQTTPublish;									// MQTTPublish FB
		MQTTPublish_SOP640_Y4: MQTT.MQTTPublish;									// MQTTPublish FB
		MQTTPublish_SOP650_KM1_2: MQTT.MQTTPublish;									// MQTTPublish FB
		MQTTPublish_SOP660_KM1_2: MQTT.MQTTPublish;									// MQTTPublish FB
		MQTTPublish_SOP670_KM1_2: MQTT.MQTTPublish;									// MQTTPublish FB
		MQTTPublish_SOP680_KM1_2: MQTT.MQTTPublish;									// MQTTPublish FB
		MQTTPublish_SOP640_RFID_Control: MQTT.MQTTPublish;							// MQTTPublish FB
		MQTTPublish_SOP640_RFID_Write: MQTT.MQTTPublish;							// MQTTPublish FB
		MQTTPublish_SOP690_RFID_Control: MQTT.MQTTPublish;							// MQTTPublish FB
		MQTTPublish_SOP690_S1: MQTT.MQTTPublish;									// MQTTPublish FB
		MQTTPublish_SOP690_S2: MQTT.MQTTPublish;									// MQTTPublish FB
		MQTTPublish_SOP690_S3: MQTT.MQTTPublish;									// MQTTPublish FB
		MQTTPublish_SOP690_S4: MQTT.MQTTPublish;									// MQTTPublish FB
		
		SOP040_K3_pTopic: WSTRING(1024):= "OP60/Actuator/SOP040_K3";						// pTopic SOP040_K3
		SOP600_H6_7_8_9_pTopic: WSTRING(1024):= "OP60/Actuator/SOP600_H6_7_8_9";			// pTopic Beacon
		SOP600_S1_pTopic: WSTRING(1024):= "OP60/Actuator/SOP600_S1";						// pTopic SOP600_S1
		SOP600_S5_pTopic: WSTRING(1024):= "OP60/Actuator/SOP600_S5";						// pTopic SOP600_S5
		SOP600_S6_pTopic: WSTRING(1024):= "OP60/Actuator/SOP600_S6";						// pTopic SOP600_S6
		SOP600_S8_pTopic: WSTRING(1024):= "OP60/Actuator/SOP600_S8";						// pTopic SOP600_S8
		SOP600_S9_pTopic: WSTRING(1024):= "OP60/Actuator/SOP600_S9";						// pTopic SOP600_S9
		SOP600_S10_pTopic: WSTRING(1024):= "OP60/Actuator/SOP600_S10";						// pTopic SOP600_S10
		SOP600_S11_pTopic: WSTRING(1024):= "OP60/Actuator/SOP600_S11";						// pTopic SOP600_S11
		SOP610_RFID_Control_pTopic: WSTRING(1024):= "OP60/SOP610/RFID_Control";				// pTopic RFID Control
		SOP610_RFID_Write_pTopic: WSTRING(1024):= "OP60/SOP610/RFID_Write";					// pTopic RFID Write
		SOP610_KM1_2_pTopic: WSTRING(1024):= "OP60/Actuator/SOP610_KM1_2";					// pTopic SOP610_KM1_2
		SOP620_KM1_2_pTopic: WSTRING(1024):= "OP60/Actuator/SOP620_KM1_2";					// pTopic SOP620_KM1_2
		SOP630_KM1_2_pTopic: WSTRING(1024):= "OP60/Actuator/SOP630_KM1_2";					// pTopic SOP630_KM1_2
		SOP640_KM1_2_pTopic: WSTRING(1024):= "OP60/Actuator/SOP640_KM1_2";					// pTopic SOP640_KM1_2
		SOP640_K2_pTopic: WSTRING(1024):= "OP60/Actuator/SOP640_K2";						// pTopic SOP640_K2
		SOP640_Y1_pTopic: WSTRING(1024):= "OP60/Actuator/SOP640_Y1";						// pTopic SOP640_Y1
		SOP640_Y2_pTopic: WSTRING(1024):= "OP60/Actuator/SOP640_Y2";						// pTopic SOP640_Y1
		SOP640_Y3_pTopic: WSTRING(1024):= "OP60/Actuator/SOP640_Y3";						// pTopic SOP640_Y1
		SOP640_Y4_pTopic: WSTRING(1024):= "OP60/Actuator/SOP640_Y4";						// pTopic SOP640_Y1
		SOP650_KM1_2_pTopic: WSTRING(1024):= "OP60/Actuator/SOP650_KM1_2";					// pTopic SOP650_KM1_2
		SOP660_KM1_2_pTopic: WSTRING(1024):= "OP60/Actuator/SOP660_KM1_2";					// pTopic SOP660_KM1_2
		SOP670_KM1_2_pTopic: WSTRING(1024):= "OP60/Actuator/SOP670_KM1_2";					// pTopic SOP670_KM1_2
		SOP680_KM1_2_pTopic: WSTRING(1024):= "OP60/Actuator/SOP680_KM1_2";					// pTopic SOP680_KM1_2
		SOP640_RFID_Control_pTopic: WSTRING(1024):= "OP60/SOP640/RFID_Control";				// pTopic RFID Control
		SOP640_RFID_Write_pTopic: WSTRING(1024):= "OP60/SOP640/RFID_Write";					// pTopic RFID Write
		SOP690_RFID_Control_pTopic: WSTRING(1024):= "OP60/SOP690/RFID_Control";				// pTopic RFID Control
		SOP690_S1_pTopic: WSTRING(1024):= "OP60/Actuator/SOP690_S1";						// pTopic SOP690_S1
		SOP690_S2_pTopic: WSTRING(1024):= "OP60/Actuator/SOP690_S2";						// pTopic SOP690_S2
		SOP690_S3_pTopic: WSTRING(1024):= "OP60/Actuator/SOP690_S3";						// pTopic SOP690_S3
		SOP690_S4_pTopic: WSTRING(1024):= "OP60/Actuator/SOP690_S4";						// pTopic SOP690_S4		

	
END_VAR
VAR // added by the converter: edge detectors and wires of the graphical bodies
    _rt1, _rt2, _rt3, _rt4, _rt5, _rt6, _rt7, _rt8, _rt9, _rt10, _rt11, _rt12, _rt13, _rt14, _rt15, _rt16, _rt17, _rt18, _rt19, _rt20, _rt21, _rt22, _rt23, _rt24, _rt25, _rt26, _rt27, _rt28, _rt29, _rt30, _rt31, _rt32, _rt33, _rt34, _rt35, _rt36, _rt37, _rt38, _rt39, _rt40, _rt41, _rt42, _rt43, _rt44, _rt45, _rt46, _rt47 : R_TRIG;
    _w1, _w2 : BOOL;
END_VAR

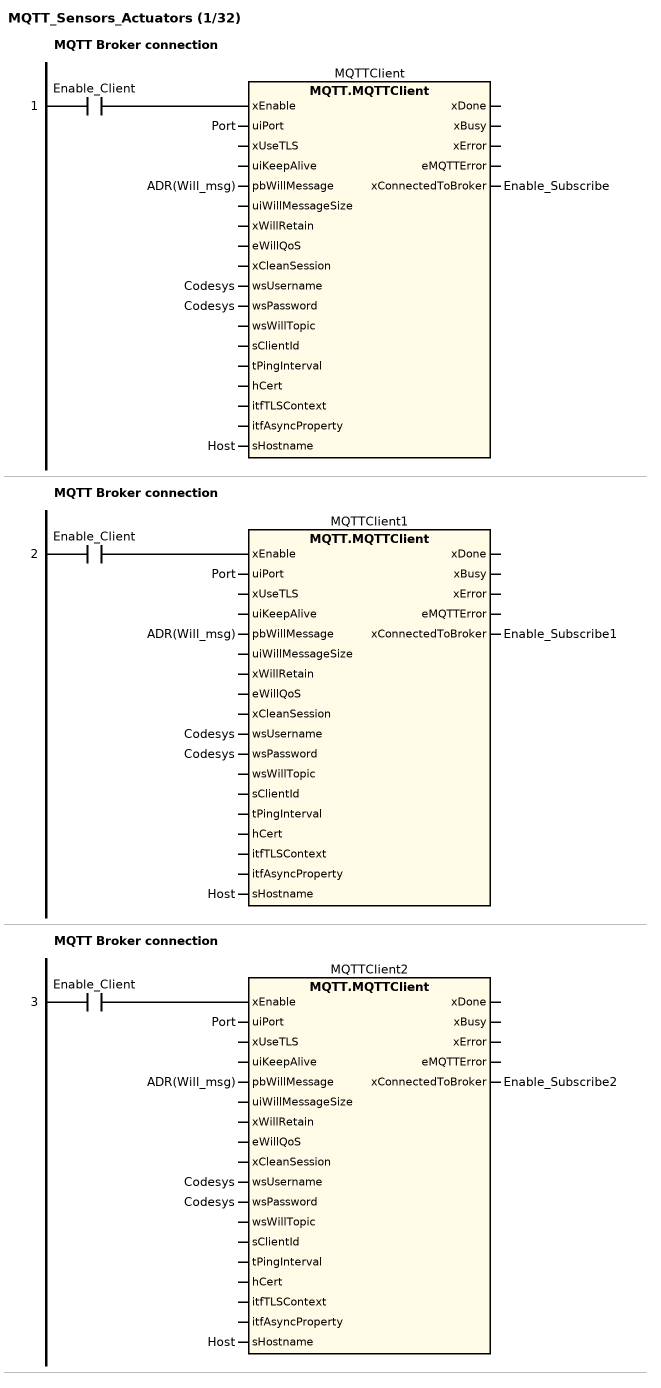
// NETWORK 1: MQTT Broker connection
MQTTClient(
    xEnable := Enable_Client,
    uiPort := Port,
    pbWillMessage := ADR(Will_msg),
    wsUsername := Codesys,
    wsPassword := Codesys,
    sHostname := Host,
    xConnectedToBroker => Enable_Subscribe); // MQTT.MQTTClient

// NETWORK 2: MQTT Broker connection
MQTTClient1(
    xEnable := Enable_Client,
    uiPort := Port,
    pbWillMessage := ADR(Will_msg),
    wsUsername := Codesys,
    wsPassword := Codesys,
    sHostname := Host,
    xConnectedToBroker => Enable_Subscribe1); // MQTT.MQTTClient

// NETWORK 3: MQTT Broker connection
MQTTClient2(
    xEnable := Enable_Client,
    uiPort := Port,
    pbWillMessage := ADR(Will_msg),
    wsUsername := Codesys,
    wsPassword := Codesys,
    sHostname := Host,
    xConnectedToBroker => Enable_Subscribe2); // MQTT.MQTTClient

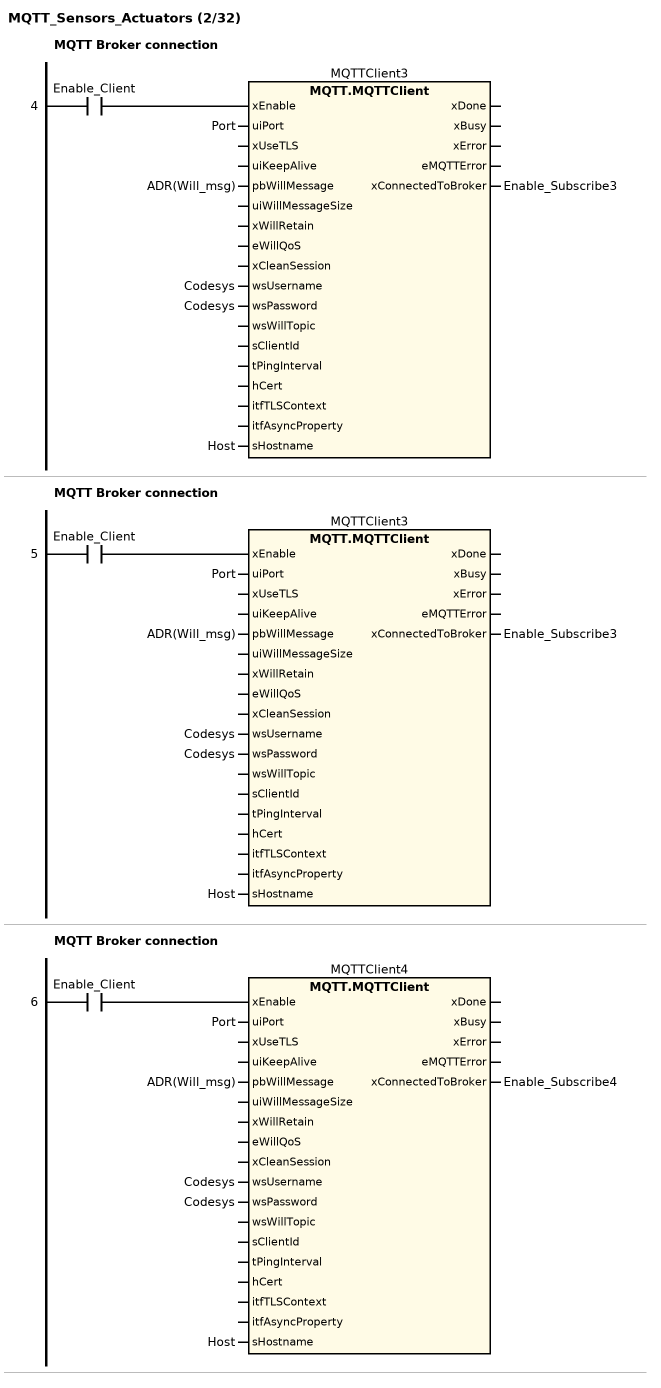
// NETWORK 4: MQTT Broker connection
MQTTClient3(
    xEnable := Enable_Client,
    uiPort := Port,
    pbWillMessage := ADR(Will_msg),
    wsUsername := Codesys,
    wsPassword := Codesys,
    sHostname := Host,
    xConnectedToBroker => Enable_Subscribe3); // MQTT.MQTTClient

// NETWORK 5: MQTT Broker connection
MQTTClient3(
    xEnable := Enable_Client,
    uiPort := Port,
    pbWillMessage := ADR(Will_msg),
    wsUsername := Codesys,
    wsPassword := Codesys,
    sHostname := Host,
    xConnectedToBroker => Enable_Subscribe3); // MQTT.MQTTClient

// NETWORK 6: MQTT Broker connection
MQTTClient4(
    xEnable := Enable_Client,
    uiPort := Port,
    pbWillMessage := ADR(Will_msg),
    wsUsername := Codesys,
    wsPassword := Codesys,
    sHostname := Host,
    xConnectedToBroker => Enable_Subscribe4); // MQTT.MQTTClient

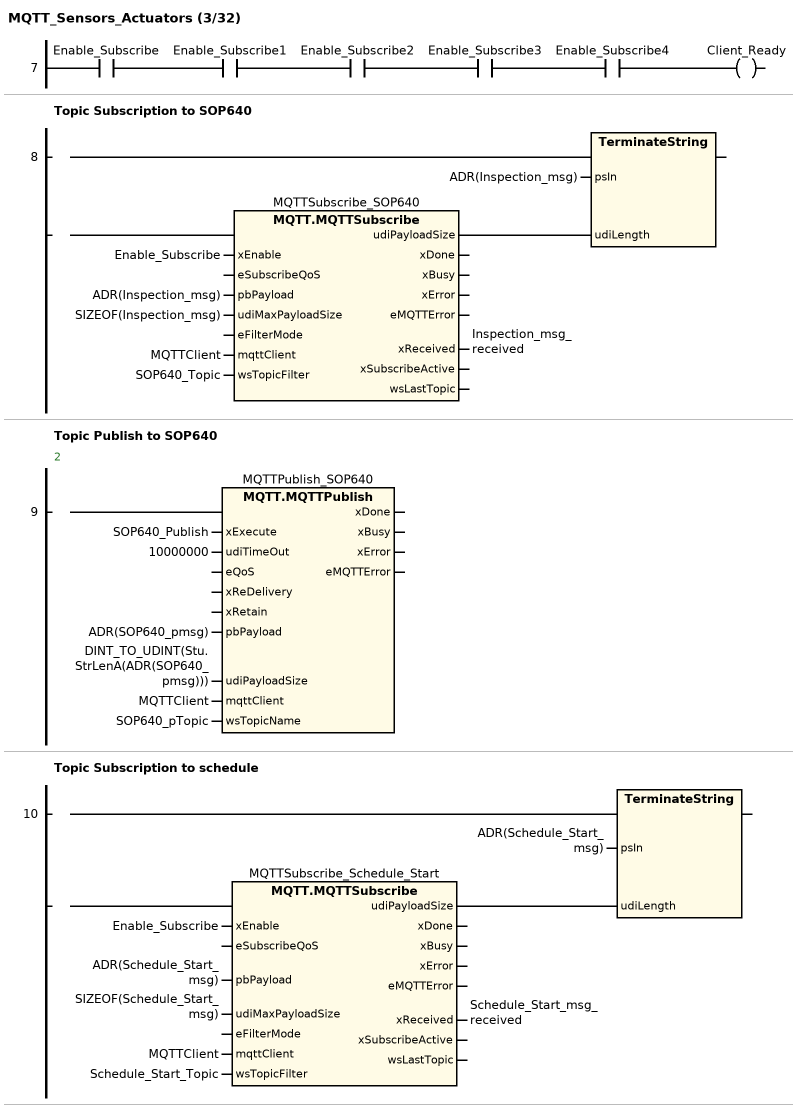
// NETWORK 7
Client_Ready := Enable_Subscribe AND Enable_Subscribe1 AND Enable_Subscribe2 AND Enable_Subscribe3 AND Enable_Subscribe4;

// NETWORK 8: Topic Subscription to SOP640
MQTTSubscribe_SOP640(
    xEnable := Enable_Subscribe,
    pbPayload := ADR(Inspection_msg),
    udiMaxPayloadSize := SIZEOF(Inspection_msg),
    mqttClient := MQTTClient,
    wsTopicFilter := SOP640_Topic,
    xReceived => Inspection_msg_received); // MQTT.MQTTSubscribe
TerminateString(psIn := ADR(Inspection_msg), udiLength := MQTTSubscribe_SOP640.udiPayloadSize);

// NETWORK 9: Topic Publish to SOP640
// 2
MQTTPublish_SOP640(
    xExecute := SOP640_Publish,
    udiTimeOut := 10000000,
    pbPayload := ADR(SOP640_pmsg),
    udiPayloadSize := DINT_TO_UDINT(Stu.StrLenA(ADR(SOP640_pmsg))),
    mqttClient := MQTTClient,
    wsTopicName := SOP640_pTopic); // MQTT.MQTTPublish

// NETWORK 10: Topic Subscription to schedule
MQTTSubscribe_Schedule_Start(
    xEnable := Enable_Subscribe,
    pbPayload := ADR(Schedule_Start_msg),
    udiMaxPayloadSize := SIZEOF(Schedule_Start_msg),
    mqttClient := MQTTClient,
    wsTopicFilter := Schedule_Start_Topic,
    xReceived => Schedule_Start_msg_received); // MQTT.MQTTSubscribe
TerminateString(psIn := ADR(Schedule_Start_msg), udiLength := MQTTSubscribe_Schedule_Start.udiPayloadSize);

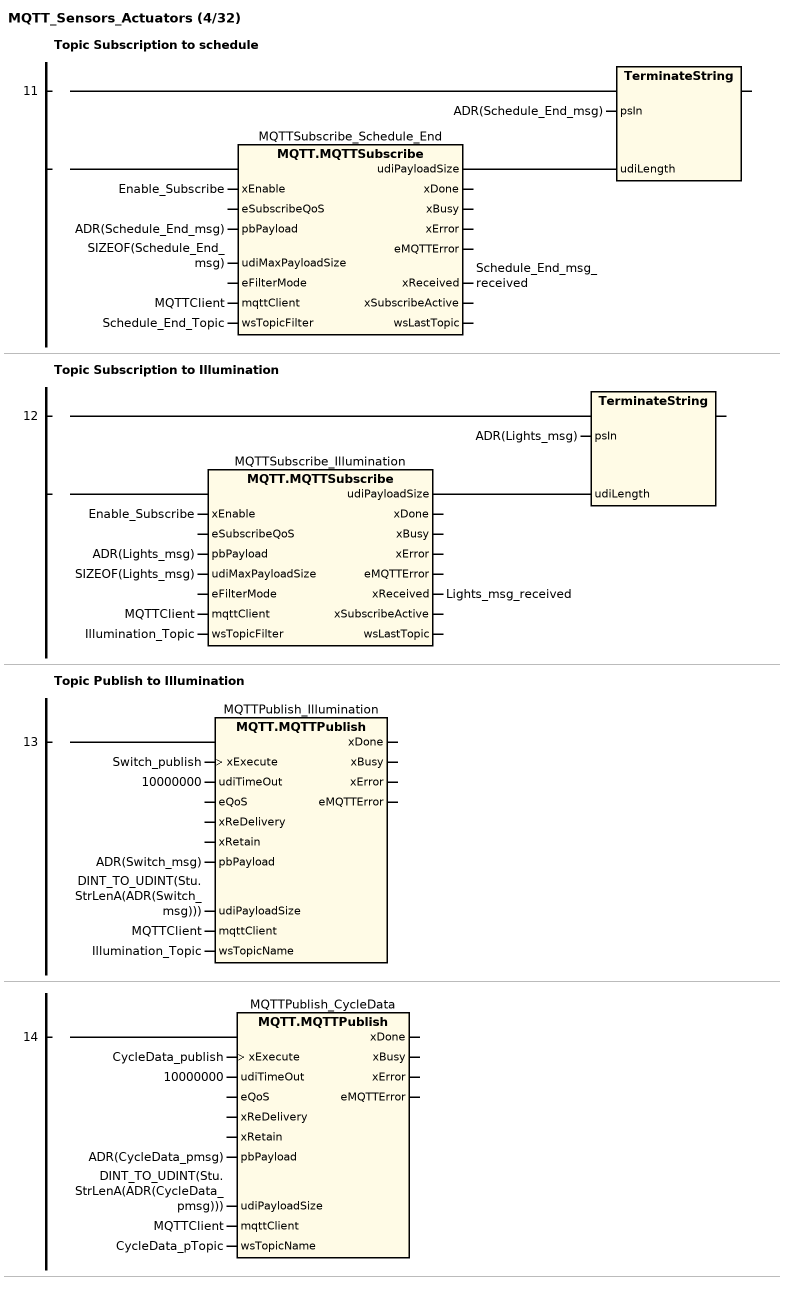
// NETWORK 11: Topic Subscription to schedule
MQTTSubscribe_Schedule_End(
    xEnable := Enable_Subscribe,
    pbPayload := ADR(Schedule_End_msg),
    udiMaxPayloadSize := SIZEOF(Schedule_End_msg),
    mqttClient := MQTTClient,
    wsTopicFilter := Schedule_End_Topic,
    xReceived => Schedule_End_msg_received); // MQTT.MQTTSubscribe
TerminateString(psIn := ADR(Schedule_End_msg), udiLength := MQTTSubscribe_Schedule_End.udiPayloadSize);

// NETWORK 12: Topic Subscription to Illumination
MQTTSubscribe_Illumination(
    xEnable := Enable_Subscribe,
    pbPayload := ADR(Lights_msg),
    udiMaxPayloadSize := SIZEOF(Lights_msg),
    mqttClient := MQTTClient,
    wsTopicFilter := Illumination_Topic,
    xReceived => Lights_msg_received); // MQTT.MQTTSubscribe
TerminateString(psIn := ADR(Lights_msg), udiLength := MQTTSubscribe_Illumination.udiPayloadSize);

// NETWORK 13: Topic Publish to Illumination
_rt1(CLK := Switch_publish);
MQTTPublish_Illumination(
    xExecute := _rt1.Q,
    udiTimeOut := 10000000,
    pbPayload := ADR(Switch_msg),
    udiPayloadSize := DINT_TO_UDINT(Stu.StrLenA(ADR(Switch_msg))),
    mqttClient := MQTTClient,
    wsTopicName := Illumination_Topic); // MQTT.MQTTPublish

// NETWORK 14
_rt2(CLK := CycleData_publish);
MQTTPublish_CycleData(
    xExecute := _rt2.Q,
    udiTimeOut := 10000000,
    pbPayload := ADR(CycleData_pmsg),
    udiPayloadSize := DINT_TO_UDINT(Stu.StrLenA(ADR(CycleData_pmsg))),
    mqttClient := MQTTClient,
    wsTopicName := CycleData_pTopic); // MQTT.MQTTPublish

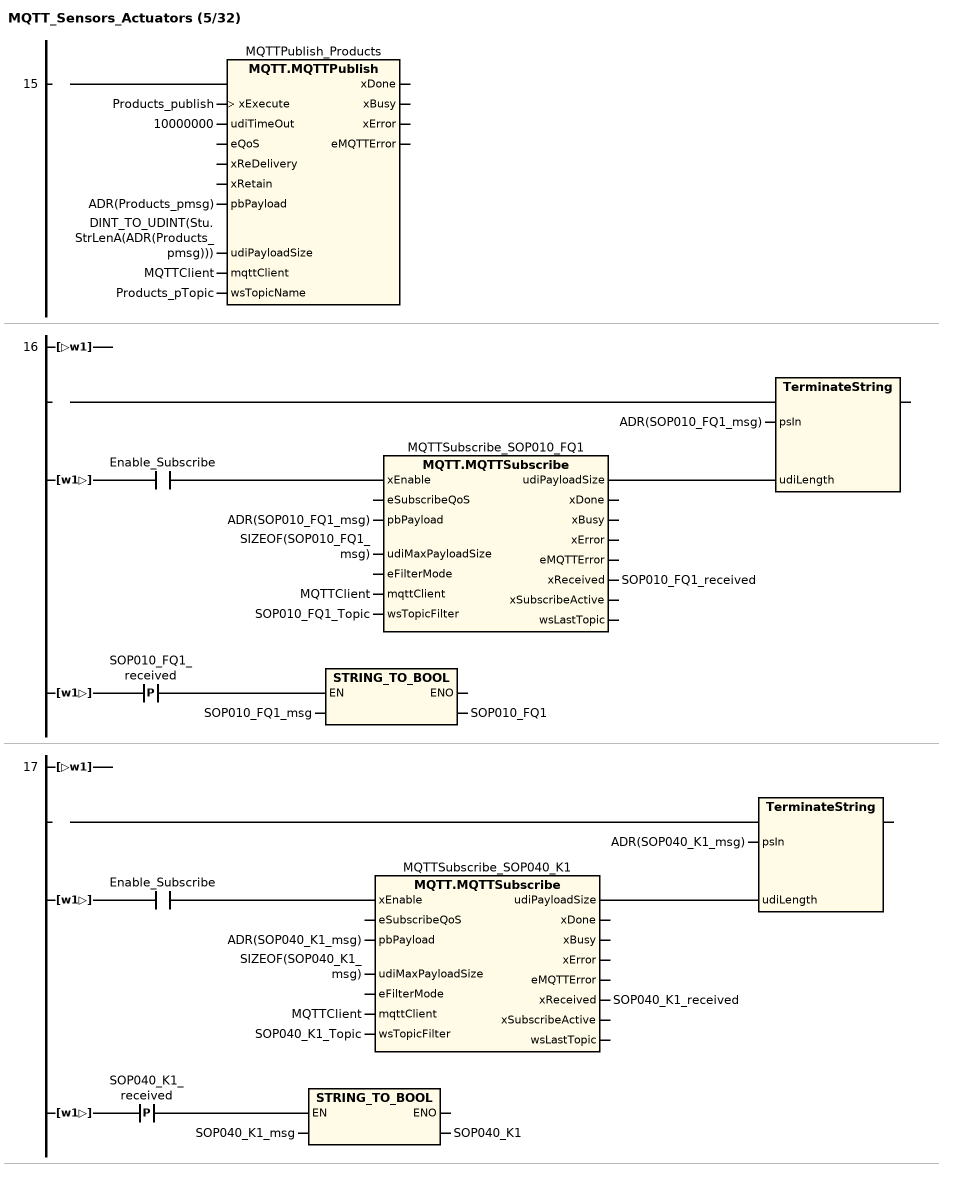
// NETWORK 15
_rt3(CLK := Products_publish);
MQTTPublish_Products(
    xExecute := _rt3.Q,
    udiTimeOut := 10000000,
    pbPayload := ADR(Products_pmsg),
    udiPayloadSize := DINT_TO_UDINT(Stu.StrLenA(ADR(Products_pmsg))),
    mqttClient := MQTTClient,
    wsTopicName := Products_pTopic); // MQTT.MQTTPublish

// NETWORK 16
MQTTSubscribe_SOP010_FQ1(
    xEnable := Enable_Subscribe,
    pbPayload := ADR(SOP010_FQ1_msg),
    udiMaxPayloadSize := SIZEOF(SOP010_FQ1_msg),
    mqttClient := MQTTClient,
    wsTopicFilter := SOP010_FQ1_Topic,
    xReceived => SOP010_FQ1_received); // MQTT.MQTTSubscribe
TerminateString(psIn := ADR(SOP010_FQ1_msg), udiLength := MQTTSubscribe_SOP010_FQ1.udiPayloadSize);
_rt4(CLK := SOP010_FQ1_received);
IF _rt4.Q THEN SOP010_FQ1 := STRING_TO_BOOL(SOP010_FQ1_msg); END_IF

// NETWORK 17
MQTTSubscribe_SOP040_K1(
    xEnable := Enable_Subscribe,
    pbPayload := ADR(SOP040_K1_msg),
    udiMaxPayloadSize := SIZEOF(SOP040_K1_msg),
    mqttClient := MQTTClient,
    wsTopicFilter := SOP040_K1_Topic,
    xReceived => SOP040_K1_received); // MQTT.MQTTSubscribe
TerminateString(psIn := ADR(SOP040_K1_msg), udiLength := MQTTSubscribe_SOP040_K1.udiPayloadSize);
_rt5(CLK := SOP040_K1_received);
IF _rt5.Q THEN SOP040_K1 := STRING_TO_BOOL(SOP040_K1_msg); END_IF

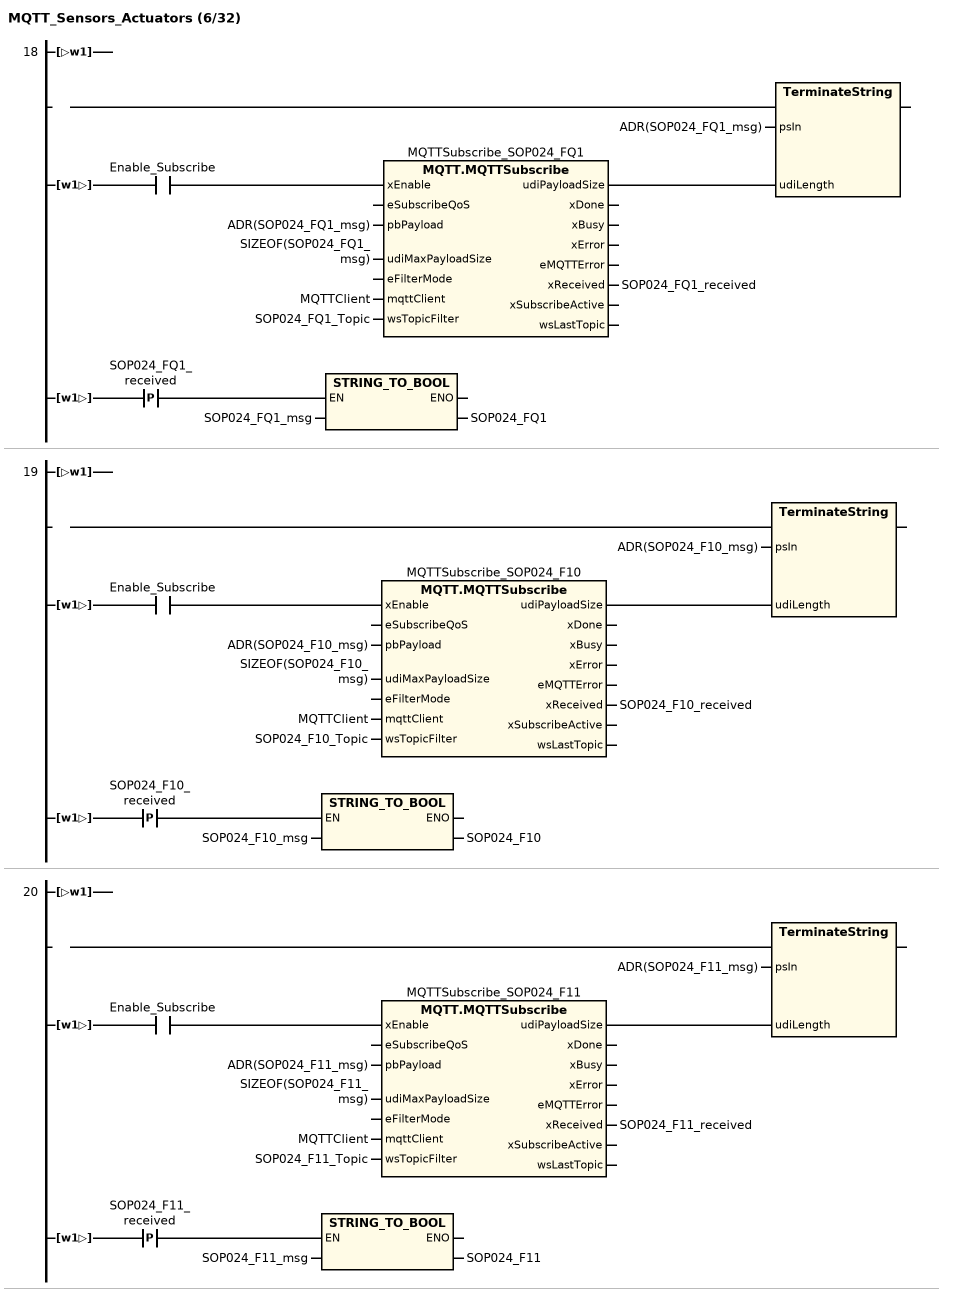
// NETWORK 18
MQTTSubscribe_SOP024_FQ1(
    xEnable := Enable_Subscribe,
    pbPayload := ADR(SOP024_FQ1_msg),
    udiMaxPayloadSize := SIZEOF(SOP024_FQ1_msg),
    mqttClient := MQTTClient,
    wsTopicFilter := SOP024_FQ1_Topic,
    xReceived => SOP024_FQ1_received); // MQTT.MQTTSubscribe
TerminateString(psIn := ADR(SOP024_FQ1_msg), udiLength := MQTTSubscribe_SOP024_FQ1.udiPayloadSize);
_rt6(CLK := SOP024_FQ1_received);
IF _rt6.Q THEN SOP024_FQ1 := STRING_TO_BOOL(SOP024_FQ1_msg); END_IF

// NETWORK 19
MQTTSubscribe_SOP024_F10(
    xEnable := Enable_Subscribe,
    pbPayload := ADR(SOP024_F10_msg),
    udiMaxPayloadSize := SIZEOF(SOP024_F10_msg),
    mqttClient := MQTTClient,
    wsTopicFilter := SOP024_F10_Topic,
    xReceived => SOP024_F10_received); // MQTT.MQTTSubscribe
TerminateString(psIn := ADR(SOP024_F10_msg), udiLength := MQTTSubscribe_SOP024_F10.udiPayloadSize);
_rt7(CLK := SOP024_F10_received);
IF _rt7.Q THEN SOP024_F10 := STRING_TO_BOOL(SOP024_F10_msg); END_IF

// NETWORK 20
MQTTSubscribe_SOP024_F11(
    xEnable := Enable_Subscribe,
    pbPayload := ADR(SOP024_F11_msg),
    udiMaxPayloadSize := SIZEOF(SOP024_F11_msg),
    mqttClient := MQTTClient,
    wsTopicFilter := SOP024_F11_Topic,
    xReceived => SOP024_F11_received); // MQTT.MQTTSubscribe
TerminateString(psIn := ADR(SOP024_F11_msg), udiLength := MQTTSubscribe_SOP024_F11.udiPayloadSize);
_rt8(CLK := SOP024_F11_received);
IF _rt8.Q THEN SOP024_F11 := STRING_TO_BOOL(SOP024_F11_msg); END_IF

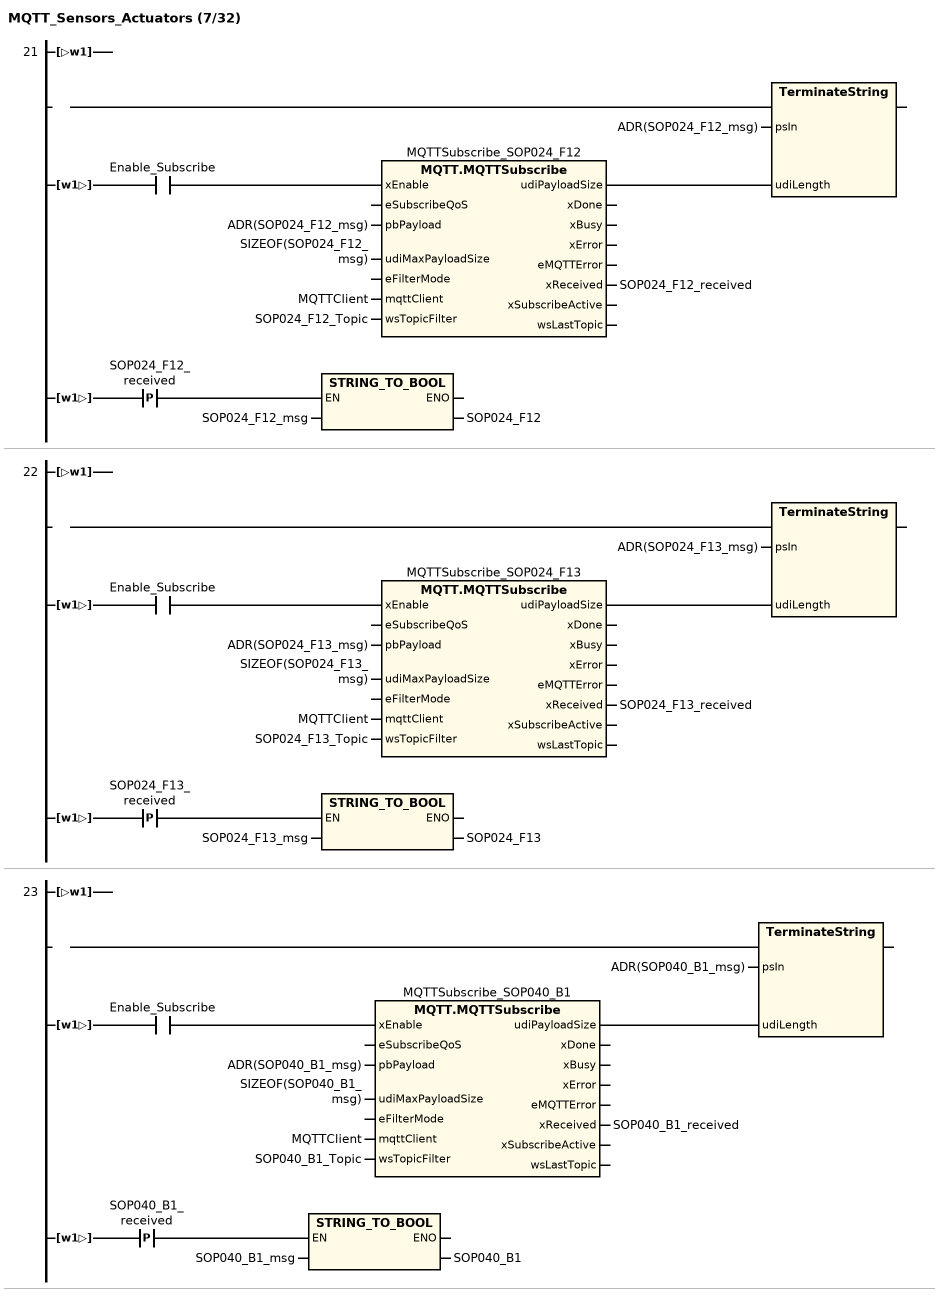
// NETWORK 21
MQTTSubscribe_SOP024_F12(
    xEnable := Enable_Subscribe,
    pbPayload := ADR(SOP024_F12_msg),
    udiMaxPayloadSize := SIZEOF(SOP024_F12_msg),
    mqttClient := MQTTClient,
    wsTopicFilter := SOP024_F12_Topic,
    xReceived => SOP024_F12_received); // MQTT.MQTTSubscribe
TerminateString(psIn := ADR(SOP024_F12_msg), udiLength := MQTTSubscribe_SOP024_F12.udiPayloadSize);
_rt9(CLK := SOP024_F12_received);
IF _rt9.Q THEN SOP024_F12 := STRING_TO_BOOL(SOP024_F12_msg); END_IF

// NETWORK 22
MQTTSubscribe_SOP024_F13(
    xEnable := Enable_Subscribe,
    pbPayload := ADR(SOP024_F13_msg),
    udiMaxPayloadSize := SIZEOF(SOP024_F13_msg),
    mqttClient := MQTTClient,
    wsTopicFilter := SOP024_F13_Topic,
    xReceived => SOP024_F13_received); // MQTT.MQTTSubscribe
TerminateString(psIn := ADR(SOP024_F13_msg), udiLength := MQTTSubscribe_SOP024_F13.udiPayloadSize);
_rt10(CLK := SOP024_F13_received);
IF _rt10.Q THEN SOP024_F13 := STRING_TO_BOOL(SOP024_F13_msg); END_IF

// NETWORK 23
MQTTSubscribe_SOP040_B1(
    xEnable := Enable_Subscribe,
    pbPayload := ADR(SOP040_B1_msg),
    udiMaxPayloadSize := SIZEOF(SOP040_B1_msg),
    mqttClient := MQTTClient,
    wsTopicFilter := SOP040_B1_Topic,
    xReceived => SOP040_B1_received); // MQTT.MQTTSubscribe
TerminateString(psIn := ADR(SOP040_B1_msg), udiLength := MQTTSubscribe_SOP040_B1.udiPayloadSize);
_rt11(CLK := SOP040_B1_received);
IF _rt11.Q THEN SOP040_B1 := STRING_TO_BOOL(SOP040_B1_msg); END_IF

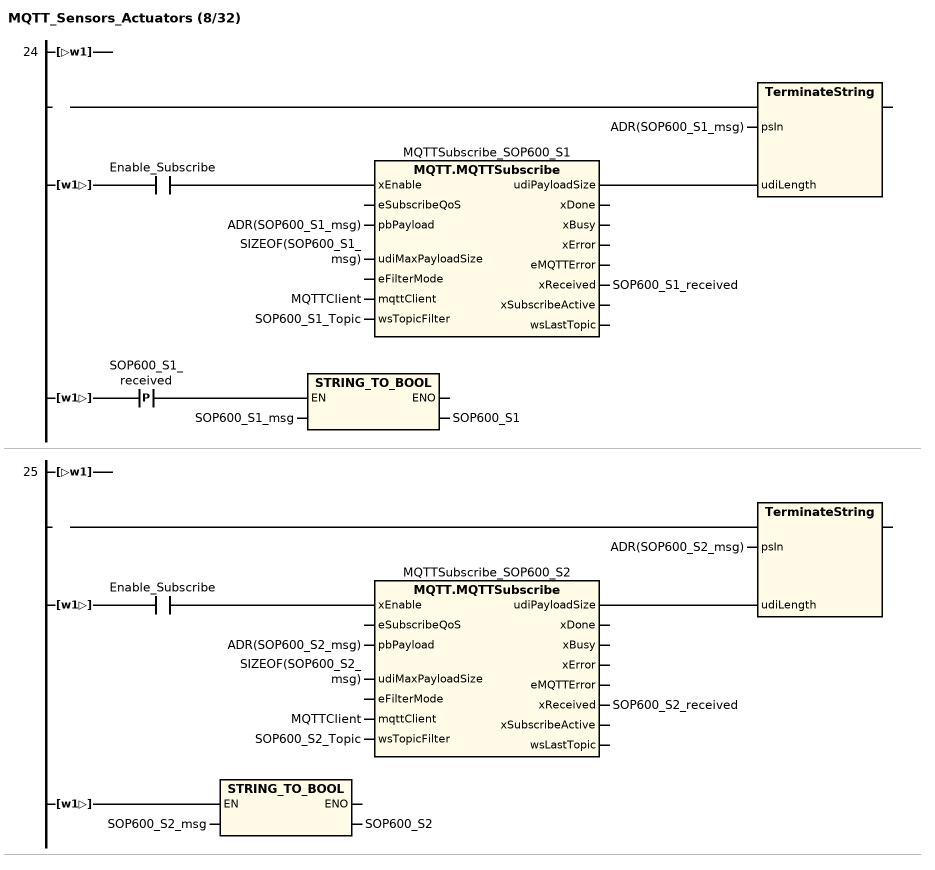
// NETWORK 24
MQTTSubscribe_SOP600_S1(
    xEnable := Enable_Subscribe,
    pbPayload := ADR(SOP600_S1_msg),
    udiMaxPayloadSize := SIZEOF(SOP600_S1_msg),
    mqttClient := MQTTClient,
    wsTopicFilter := SOP600_S1_Topic,
    xReceived => SOP600_S1_received); // MQTT.MQTTSubscribe
TerminateString(psIn := ADR(SOP600_S1_msg), udiLength := MQTTSubscribe_SOP600_S1.udiPayloadSize);
_rt12(CLK := SOP600_S1_received);
IF _rt12.Q THEN SOP600_S1 := STRING_TO_BOOL(SOP600_S1_msg); END_IF

// NETWORK 25
MQTTSubscribe_SOP600_S2(
    xEnable := Enable_Subscribe,
    pbPayload := ADR(SOP600_S2_msg),
    udiMaxPayloadSize := SIZEOF(SOP600_S2_msg),
    mqttClient := MQTTClient,
    wsTopicFilter := SOP600_S2_Topic,
    xReceived => SOP600_S2_received); // MQTT.MQTTSubscribe
TerminateString(psIn := ADR(SOP600_S2_msg), udiLength := MQTTSubscribe_SOP600_S2.udiPayloadSize);
SOP600_S2 := STRING_TO_BOOL(SOP600_S2_msg);

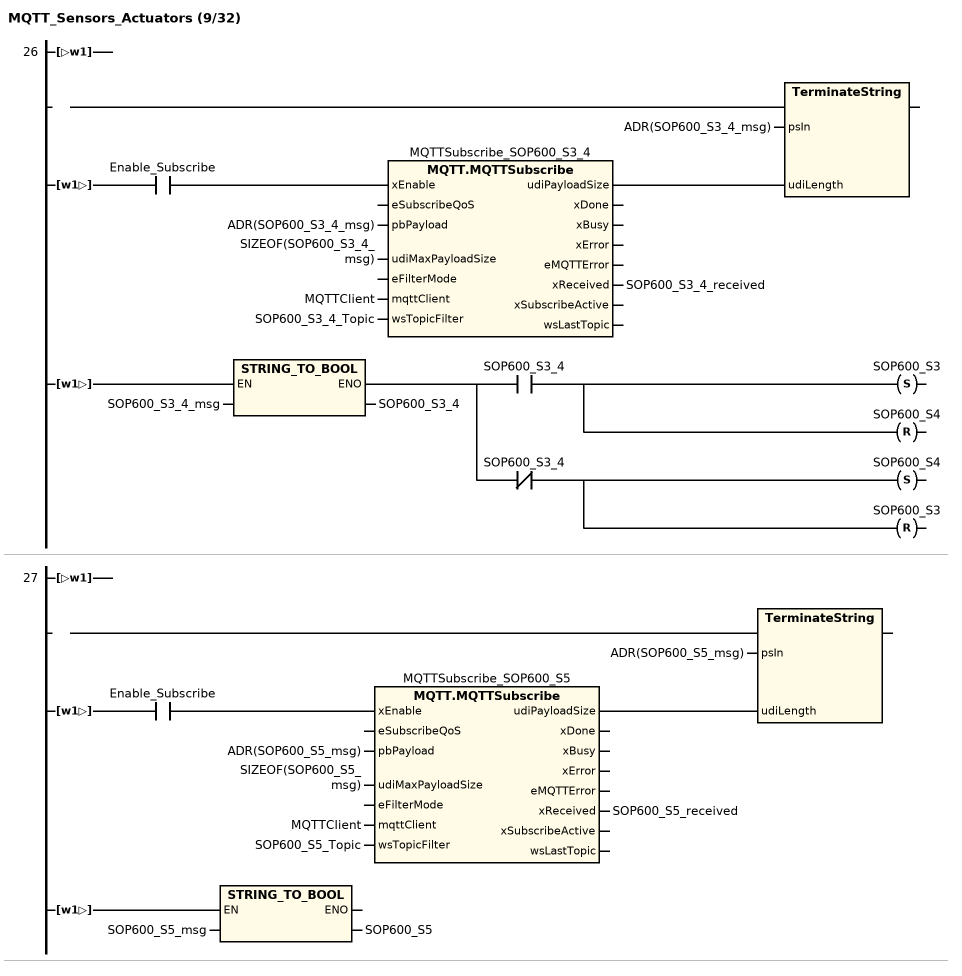
// NETWORK 26
MQTTSubscribe_SOP600_S3_4(
    xEnable := Enable_Subscribe,
    pbPayload := ADR(SOP600_S3_4_msg),
    udiMaxPayloadSize := SIZEOF(SOP600_S3_4_msg),
    mqttClient := MQTTClient,
    wsTopicFilter := SOP600_S3_4_Topic,
    xReceived => SOP600_S3_4_received); // MQTT.MQTTSubscribe
TerminateString(psIn := ADR(SOP600_S3_4_msg), udiLength := MQTTSubscribe_SOP600_S3_4.udiPayloadSize);
SOP600_S3_4 := STRING_TO_BOOL(SOP600_S3_4_msg);
_w1 := SOP600_S3_4;
SOP600_S3 S= _w1;
SOP600_S4 R= _w1;
_w2 := NOT SOP600_S3_4;
SOP600_S4 S= _w2;
SOP600_S3 R= _w2;

// NETWORK 27
MQTTSubscribe_SOP600_S5(
    xEnable := Enable_Subscribe,
    pbPayload := ADR(SOP600_S5_msg),
    udiMaxPayloadSize := SIZEOF(SOP600_S5_msg),
    mqttClient := MQTTClient,
    wsTopicFilter := SOP600_S5_Topic,
    xReceived => SOP600_S5_received); // MQTT.MQTTSubscribe
TerminateString(psIn := ADR(SOP600_S5_msg), udiLength := MQTTSubscribe_SOP600_S5.udiPayloadSize);
SOP600_S5 := STRING_TO_BOOL(SOP600_S5_msg);

